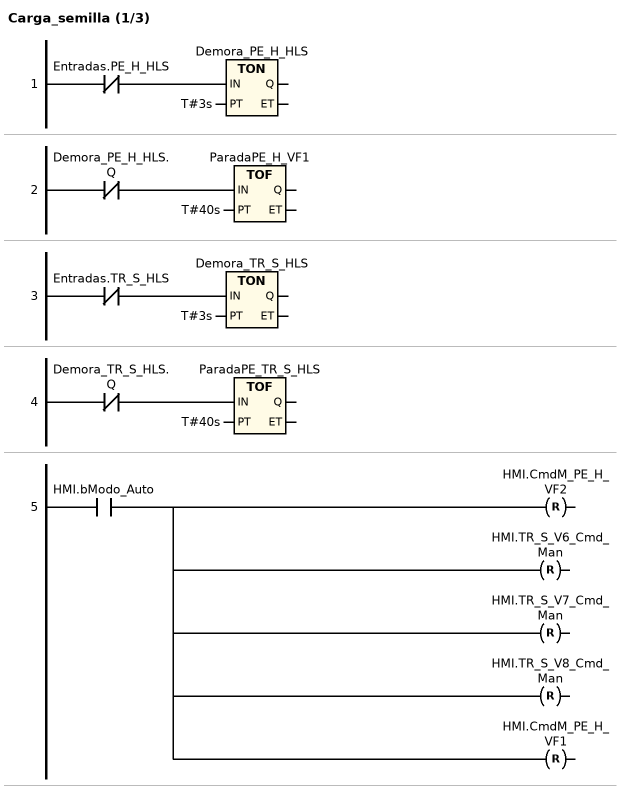
// NETWORK 1
Demora_PE_H_HLS(IN := NOT Entradas.PE_H_HLS, PT := T#3s); // TON

// NETWORK 2
ParadaPE_H_VF1(IN := NOT Demora_PE_H_HLS.Q, PT := T#40s); // TOF

// NETWORK 3
Demora_TR_S_HLS(IN := NOT Entradas.TR_S_HLS, PT := T#3s); // TON

// NETWORK 4
ParadaPE_TR_S_HLS(IN := NOT Demora_TR_S_HLS.Q, PT := T#40s); // TOF

// NETWORK 5
_w1 := HMI.bModo_Auto;
HMI.CmdM_PE_H_VF2 R= _w1;
HMI.TR_S_V6_Cmd_Man R= _w1;
HMI.TR_S_V7_Cmd_Man R= _w1;
HMI.TR_S_V8_Cmd_Man R= _w1;
HMI.CmdM_PE_H_VF1 R= _w1;

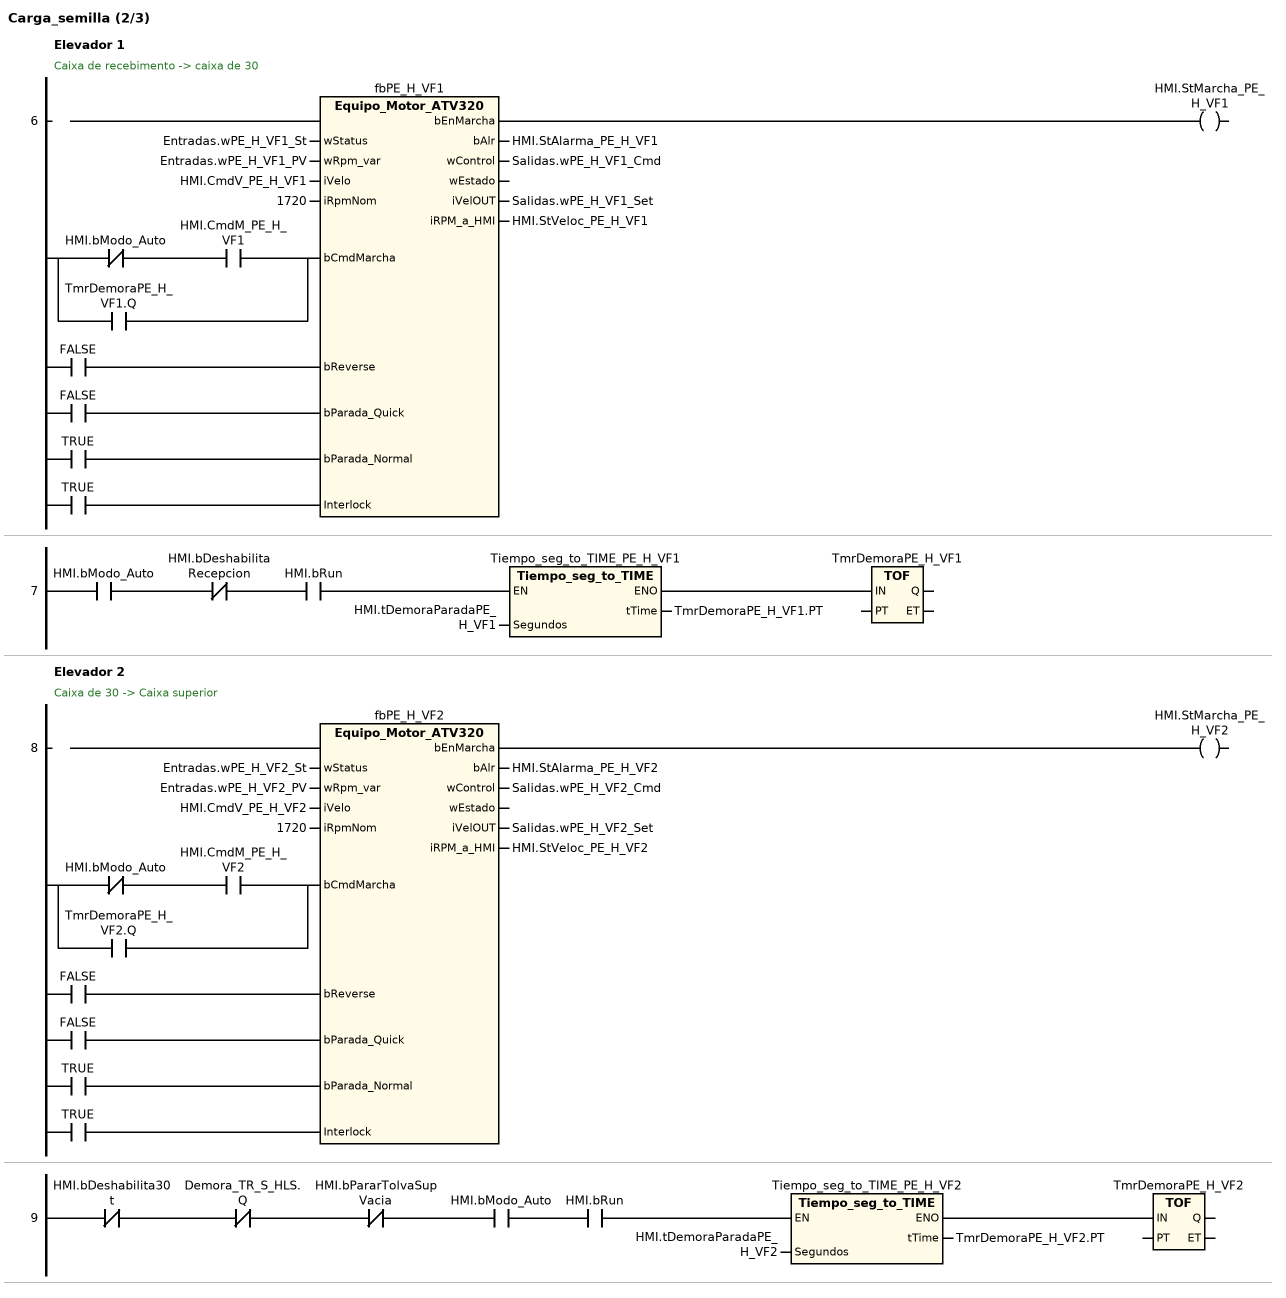
// NETWORK 6: Elevador 1
// Caixa de recebimento -> caixa de 30
fbPE_H_VF1(
    wStatus := Entradas.wPE_H_VF1_St,
    wRpm_var := Entradas.wPE_H_VF1_PV,
    iVelo := HMI.CmdV_PE_H_VF1,
    iRpmNom := 1720,
    bCmdMarcha := NOT HMI.bModo_Auto AND HMI.CmdM_PE_H_VF1 OR TmrDemoraPE_H_VF1.Q,
    bReverse := FALSE,
    bParada_Quick := FALSE,
    bParada_Normal := TRUE,
    Interlock := TRUE,
    bAlr => HMI.StAlarma_PE_H_VF1,
    wControl => Salidas.wPE_H_VF1_Cmd,
    iVelOUT => Salidas.wPE_H_VF1_Set,
    iRPM_a_HMI => HMI.StVeloc_PE_H_VF1); // Equipo_Motor_ATV320
HMI.StMarcha_PE_H_VF1 := fbPE_H_VF1.bEnMarcha;

// NETWORK 7
_w2 := HMI.bModo_Auto AND NOT HMI.bDeshabilitaRecepcion AND HMI.bRun;
IF _w2 THEN
    Tiempo_seg_to_TIME_PE_H_VF1(Segundos := HMI.tDemoraParadaPE_H_VF1, tTime => TmrDemoraPE_H_VF1.PT); // Tiempo_seg_to_TIME
END_IF
TmrDemoraPE_H_VF1(IN := _w2); // TOF

// NETWORK 8: Elevador 2
// Caixa de 30 -> Caixa superior
fbPE_H_VF2(
    wStatus := Entradas.wPE_H_VF2_St,
    wRpm_var := Entradas.wPE_H_VF2_PV,
    iVelo := HMI.CmdV_PE_H_VF2,
    iRpmNom := 1720,
    bCmdMarcha := NOT HMI.bModo_Auto AND HMI.CmdM_PE_H_VF2 OR TmrDemoraPE_H_VF2.Q,
    bReverse := FALSE,
    bParada_Quick := FALSE,
    bParada_Normal := TRUE,
    Interlock := TRUE,
    bAlr => HMI.StAlarma_PE_H_VF2,
    wControl => Salidas.wPE_H_VF2_Cmd,
    iVelOUT => Salidas.wPE_H_VF2_Set,
    iRPM_a_HMI => HMI.StVeloc_PE_H_VF2); // Equipo_Motor_ATV320
HMI.StMarcha_PE_H_VF2 := fbPE_H_VF2.bEnMarcha;

// NETWORK 9
_w3 := NOT HMI.bDeshabilita30t AND NOT Demora_TR_S_HLS.Q AND NOT HMI.bPararTolvaSupVacia AND HMI.bModo_Auto AND HMI.bRun;
IF _w3 THEN
    Tiempo_seg_to_TIME_PE_H_VF2(Segundos := HMI.tDemoraParadaPE_H_VF2, tTime => TmrDemoraPE_H_VF2.PT); // Tiempo_seg_to_TIME
END_IF
TmrDemoraPE_H_VF2(IN := _w3); // TOF

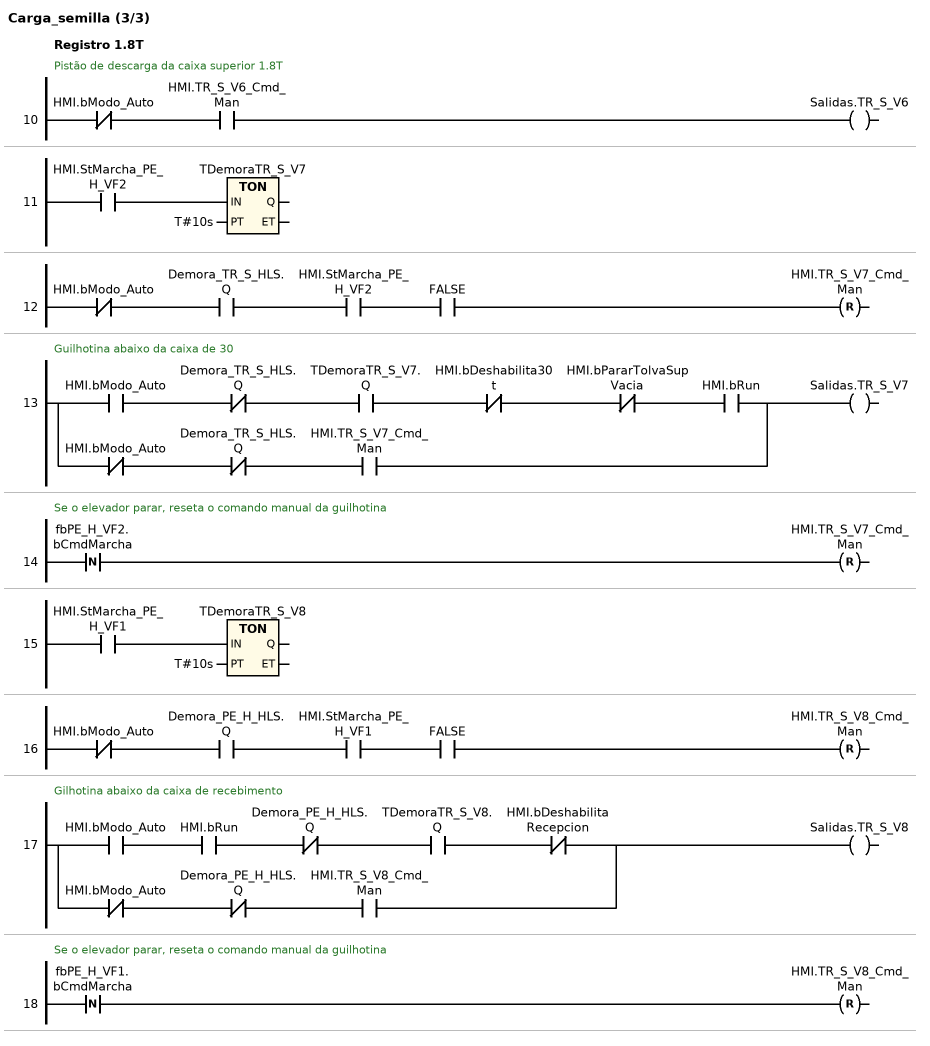
// NETWORK 10: Registro 1.8T
// Pistão de descarga da caixa superior 1.8T
Salidas.TR_S_V6 := NOT HMI.bModo_Auto AND HMI.TR_S_V6_Cmd_Man;

// NETWORK 11
TDemoraTR_S_V7(IN := HMI.StMarcha_PE_H_VF2, PT := T#10s); // TON

// NETWORK 12
HMI.TR_S_V7_Cmd_Man R= NOT HMI.bModo_Auto AND Demora_TR_S_HLS.Q AND HMI.StMarcha_PE_H_VF2 AND FALSE;

// NETWORK 13
// Guilhotina abaixo da caixa de 30
Salidas.TR_S_V7 := HMI.bModo_Auto AND NOT Demora_TR_S_HLS.Q AND TDemoraTR_S_V7.Q AND NOT HMI.bDeshabilita30t AND NOT HMI.bPararTolvaSupVacia AND HMI.bRun OR NOT HMI.bModo_Auto AND NOT Demora_TR_S_HLS.Q AND HMI.TR_S_V7_Cmd_Man;

// NETWORK 14
// Se o elevador parar, reseta o comando manual da guilhotina
_ft1(CLK := fbPE_H_VF2.bCmdMarcha);
HMI.TR_S_V7_Cmd_Man R= _ft1.Q;

// NETWORK 15
TDemoraTR_S_V8(IN := HMI.StMarcha_PE_H_VF1, PT := T#10s); // TON

// NETWORK 16
HMI.TR_S_V8_Cmd_Man R= NOT HMI.bModo_Auto AND Demora_PE_H_HLS.Q AND HMI.StMarcha_PE_H_VF1 AND FALSE;

// NETWORK 17
// Gilhotina abaixo da caixa de recebimento
Salidas.TR_S_V8 := HMI.bModo_Auto AND HMI.bRun AND NOT Demora_PE_H_HLS.Q AND TDemoraTR_S_V8.Q AND NOT HMI.bDeshabilitaRecepcion OR NOT HMI.bModo_Auto AND NOT Demora_PE_H_HLS.Q AND HMI.TR_S_V8_Cmd_Man;

// NETWORK 18
// Se o elevador parar, reseta o comando manual da guilhotina
_ft2(CLK := fbPE_H_VF1.bCmdMarcha);
HMI.TR_S_V8_Cmd_Man R= _ft2.Q;

END_PROGRAM

// ---- POUs/Polvo 1/Dosificador_Polvo_1.TcPOU
PROGRAM Dosificador_Polvo_1
VAR
	fbDosificador_P1 :Equipo_Motor_ATV320;
	Balanza_P1_WT1: Balanza;
	fbTR_P1_VI: Equipo_Motor_ATV320;
	TararP1:BOOL;
	dHS:DINT;
	
	Tmr_Alr_ZeroSpeed: TON;
	TDemoraInyectarPolvo: TON;
	Tiempo_seg_to_TIME_TDemoraInyec: Tiempo_seg_to_TIME;
	Auxtdemora: TIME;
	Calc_Veloc_Polvo_1: Calc_Veloc_Polvo;
	Calc_Veloc_Polvo_1i: Calc_Veloc_Polvo;
	Tiempo_seg_to_TIME_TInyeccion: Tiempo_seg_to_TIME;
	AuxInyec: TIME;
	TInyeccion: TON;
	ModoCalibrarP1 :BOOL;
	
	InyectarCalibrarP1: BOOL;
	Calibracion_Po_calc_P1: Calibracion_Po_calc;
	PolvoAsociado:STRING;
	TR_P1_WT1_rValue_REAL: REAL;
	TON_SolicitaPo: TON;
END_VAR
VAR PERSISTENT
	UltimaCalibracao	:UDINT;	//Data da ultima calibração feita com sucesso
END_VAR
VAR // added by the converter: edge detectors and wires of the graphical bodies
    _w1, _w2, _w3 : BOOL;
    _ft1 : F_TRIG;
    _rt1 : R_TRIG;
END_VAR

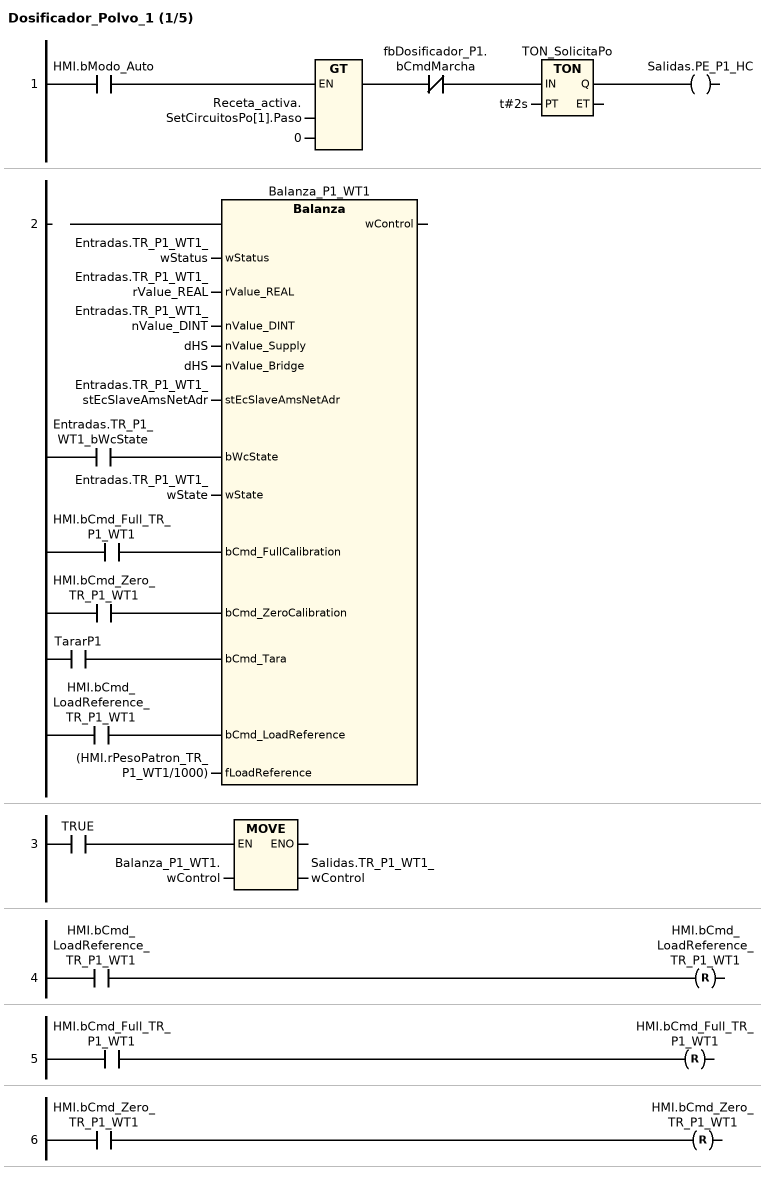
// NETWORK 1
TON_SolicitaPo(IN := (HMI.bModo_Auto AND Receta_activa.SetCircuitosPo[1].Paso > 0) AND NOT fbDosificador_P1.bCmdMarcha, PT := t#2s); // TON
Salidas.PE_P1_HC := TON_SolicitaPo.Q;

// NETWORK 2
Balanza_P1_WT1(
    wStatus := Entradas.TR_P1_WT1_wStatus,
    rValue_REAL := Entradas.TR_P1_WT1_rValue_REAL,
    nValue_DINT := Entradas.TR_P1_WT1_nValue_DINT,
    nValue_Supply := dHS,
    nValue_Bridge := dHS,
    stEcSlaveAmsNetAdr := Entradas.TR_P1_WT1_stEcSlaveAmsNetAdr,
    bWcState := Entradas.TR_P1_WT1_bWcState,
    wState := Entradas.TR_P1_WT1_wState,
    bCmd_FullCalibration := HMI.bCmd_Full_TR_P1_WT1,
    bCmd_ZeroCalibration := HMI.bCmd_Zero_TR_P1_WT1,
    bCmd_Tara := TararP1,
    bCmd_LoadReference := HMI.bCmd_LoadReference_TR_P1_WT1,
    fLoadReference := (HMI.rPesoPatron_TR_P1_WT1/1000)); // Balanza

// NETWORK 3
Salidas.TR_P1_WT1_wControl := Balanza_P1_WT1.wControl;

// NETWORK 4
HMI.bCmd_LoadReference_TR_P1_WT1 R= HMI.bCmd_LoadReference_TR_P1_WT1;

// NETWORK 5
HMI.bCmd_Full_TR_P1_WT1 R= HMI.bCmd_Full_TR_P1_WT1;

// NETWORK 6
HMI.bCmd_Zero_TR_P1_WT1 R= HMI.bCmd_Zero_TR_P1_WT1;

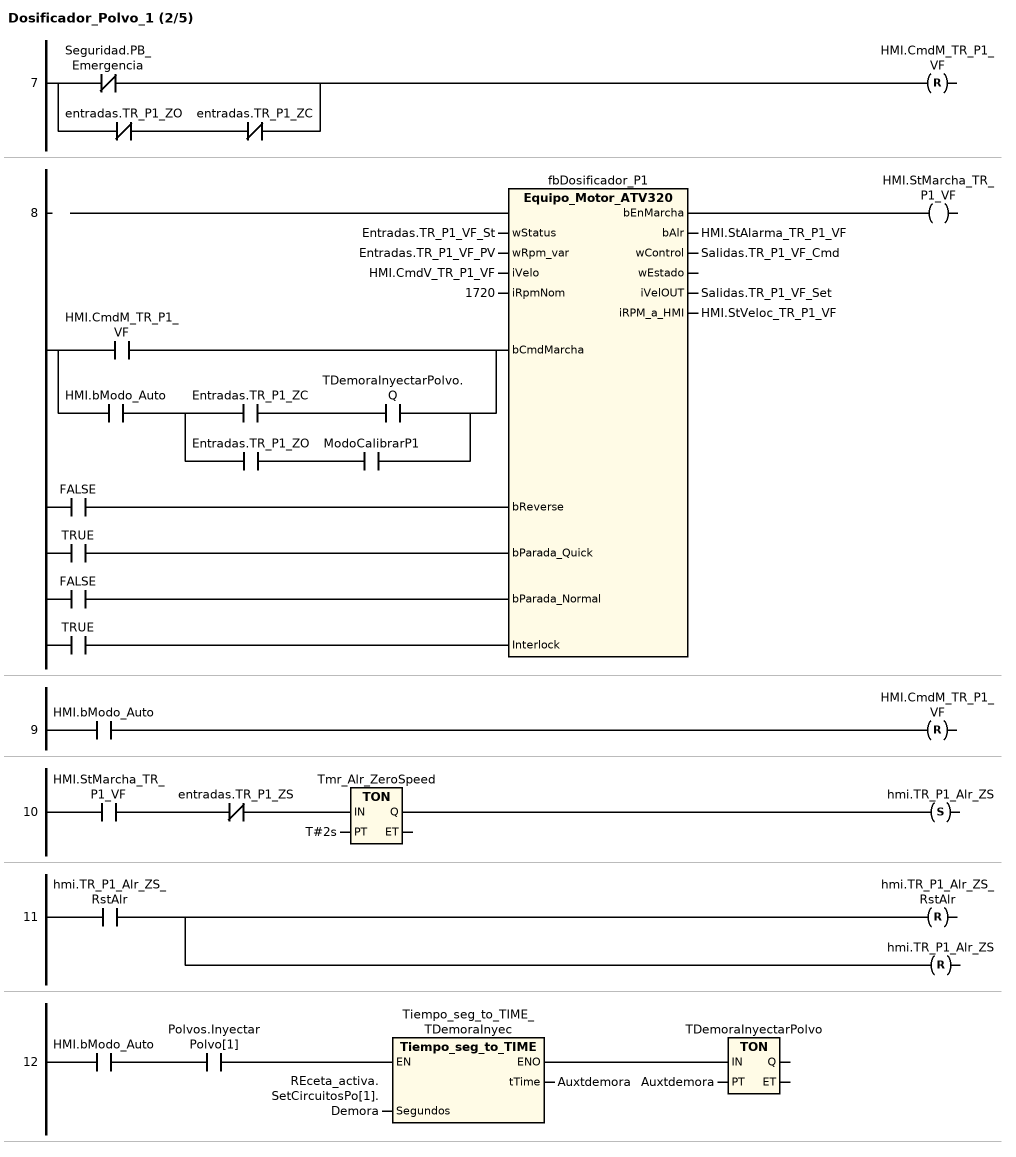
// NETWORK 7
HMI.CmdM_TR_P1_VF R= NOT Seguridad.PB_Emergencia OR NOT entradas.TR_P1_ZO AND NOT entradas.TR_P1_ZC;

// NETWORK 8
fbDosificador_P1(
    wStatus := Entradas.TR_P1_VF_St,
    wRpm_var := Entradas.TR_P1_VF_PV,
    iVelo := HMI.CmdV_TR_P1_VF,
    iRpmNom := 1720,
    bCmdMarcha := HMI.CmdM_TR_P1_VF OR HMI.bModo_Auto AND (Entradas.TR_P1_ZC AND TDemoraInyectarPolvo.Q OR Entradas.TR_P1_ZO AND ModoCalibrarP1),
    bReverse := FALSE,
    bParada_Quick := TRUE,
    bParada_Normal := FALSE,
    Interlock := TRUE,
    bAlr => HMI.StAlarma_TR_P1_VF,
    wControl => Salidas.TR_P1_VF_Cmd,
    iVelOUT => Salidas.TR_P1_VF_Set,
    iRPM_a_HMI => HMI.StVeloc_TR_P1_VF); // Equipo_Motor_ATV320
HMI.StMarcha_TR_P1_VF := fbDosificador_P1.bEnMarcha;

// NETWORK 9
HMI.CmdM_TR_P1_VF R= HMI.bModo_Auto;

// NETWORK 10
Tmr_Alr_ZeroSpeed(IN := HMI.StMarcha_TR_P1_VF AND NOT entradas.TR_P1_ZS, PT := T#2s); // TON
hmi.TR_P1_Alr_ZS S= Tmr_Alr_ZeroSpeed.Q;

// NETWORK 11
_w1 := hmi.TR_P1_Alr_ZS_RstAlr;
hmi.TR_P1_Alr_ZS_RstAlr R= _w1;
hmi.TR_P1_Alr_ZS R= _w1;

// NETWORK 12
_w2 := HMI.bModo_Auto AND Polvos.InyectarPolvo[1];
IF _w2 THEN
    Tiempo_seg_to_TIME_TDemoraInyec(Segundos := REceta_activa.SetCircuitosPo[1].Demora, tTime => Auxtdemora); // Tiempo_seg_to_TIME
END_IF
TDemoraInyectarPolvo(IN := _w2, PT := Auxtdemora); // TON

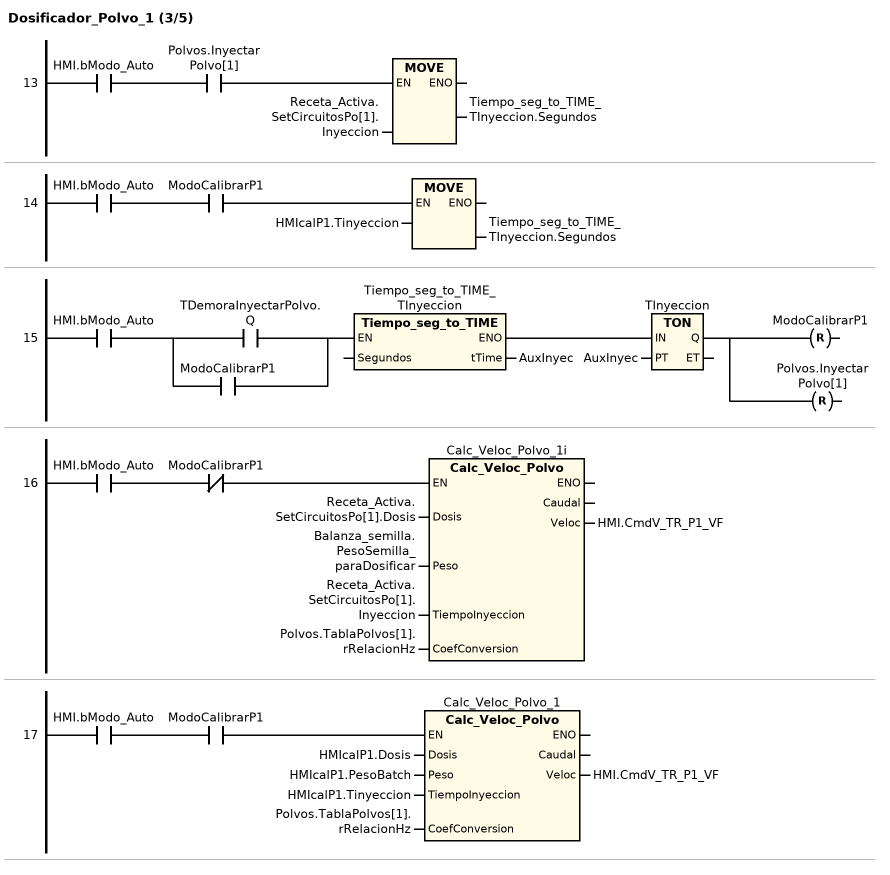
// NETWORK 13
IF HMI.bModo_Auto AND Polvos.InyectarPolvo[1] THEN
    Tiempo_seg_to_TIME_TInyeccion.Segundos := Receta_Activa.SetCircuitosPo[1].Inyeccion;
END_IF

// NETWORK 14
IF HMI.bModo_Auto AND ModoCalibrarP1 THEN Tiempo_seg_to_TIME_TInyeccion.Segundos := HMIcalP1.Tinyeccion; END_IF

// NETWORK 15
_w3 := HMI.bModo_Auto AND (TDemoraInyectarPolvo.Q OR ModoCalibrarP1);
IF _w3 THEN
    Tiempo_seg_to_TIME_TInyeccion(tTime => AuxInyec); // Tiempo_seg_to_TIME
END_IF
TInyeccion(IN := _w3, PT := AuxInyec); // TON
ModoCalibrarP1 R= TInyeccion.Q;
Polvos.InyectarPolvo[1] R= TInyeccion.Q;

// NETWORK 16
IF HMI.bModo_Auto AND NOT ModoCalibrarP1 THEN
    Calc_Veloc_Polvo_1i(
        Dosis := Receta_Activa.SetCircuitosPo[1].Dosis,
        Peso := Balanza_semilla.PesoSemilla_paraDosificar,
        TiempoInyeccion := Receta_Activa.SetCircuitosPo[1].Inyeccion,
        CoefConversion := Polvos.TablaPolvos[1].rRelacionHz,
        Veloc => HMI.CmdV_TR_P1_VF); // Calc_Veloc_Polvo
END_IF

// NETWORK 17
IF HMI.bModo_Auto AND ModoCalibrarP1 THEN
    Calc_Veloc_Polvo_1(
        Dosis := HMIcalP1.Dosis,
        Peso := HMIcalP1.PesoBatch,
        TiempoInyeccion := HMIcalP1.Tinyeccion,
        CoefConversion := Polvos.TablaPolvos[1].rRelacionHz,
        Veloc => HMI.CmdV_TR_P1_VF); // Calc_Veloc_Polvo
END_IF

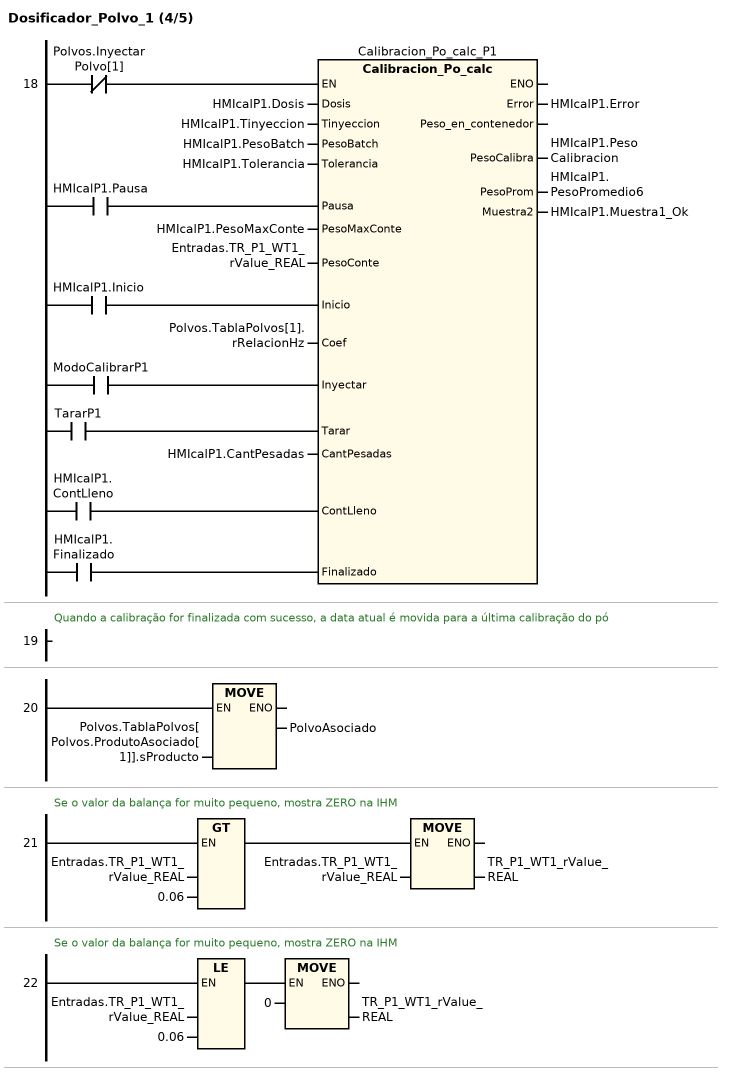
// NETWORK 18
IF NOT Polvos.InyectarPolvo[1] THEN
    Calibracion_Po_calc_P1(
        Dosis := HMIcalP1.Dosis,
        Tinyeccion := HMIcalP1.Tinyeccion,
        PesoBatch := HMIcalP1.PesoBatch,
        Tolerancia := HMIcalP1.Tolerancia,
        Pausa := HMIcalP1.Pausa,
        PesoMaxConte := HMIcalP1.PesoMaxConte,
        PesoConte := Entradas.TR_P1_WT1_rValue_REAL,
        Inicio := HMIcalP1.Inicio,
        Coef := Polvos.TablaPolvos[1].rRelacionHz,
        Inyectar := ModoCalibrarP1,
        Tarar := TararP1,
        CantPesadas := HMIcalP1.CantPesadas,
        ContLleno := HMIcalP1.ContLleno,
        Finalizado := HMIcalP1.Finalizado,
        Error => HMIcalP1.Error,
        PesoCalibra => HMIcalP1.PesoCalibracion,
        PesoProm => HMIcalP1.PesoPromedio6,
        Muestra2 => HMIcalP1.Muestra1_Ok); // Calibracion_Po_calc
END_IF

// NETWORK 19
// Quando a calibração for finalizada com sucesso, a data atual é movida para a última calibração do pó

// NETWORK 20
PolvoAsociado := Polvos.TablaPolvos[Polvos.ProdutoAsociado[1]].sProducto;

// NETWORK 21
// Se o valor da balança for muito pequeno, mostra ZERO na IHM
IF Entradas.TR_P1_WT1_rValue_REAL > 0.06 THEN TR_P1_WT1_rValue_REAL := Entradas.TR_P1_WT1_rValue_REAL; END_IF

// NETWORK 22
// Se o valor da balança for muito pequeno, mostra ZERO na IHM
IF Entradas.TR_P1_WT1_rValue_REAL <= 0.06 THEN TR_P1_WT1_rValue_REAL := 0; END_IF

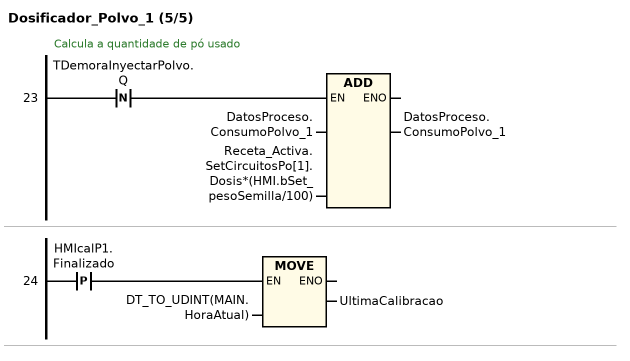
// NETWORK 23
// Calcula a quantidade de pó usado
_ft1(CLK := TDemoraInyectarPolvo.Q);
IF _ft1.Q THEN
    DatosProceso.ConsumoPolvo_1 := DatosProceso.ConsumoPolvo_1 + (Receta_Activa.SetCircuitosPo[1].Dosis*(HMI.bSet_pesoSemilla/100));
END_IF

// NETWORK 24
_rt1(CLK := HMIcalP1.Finalizado);
IF _rt1.Q THEN UltimaCalibracao := DT_TO_UDINT(MAIN.HoraAtual); END_IF

END_PROGRAM

// ---- POUs/Elementos/Calc_Veloc_Polvo.TcPOU
FUNCTION_BLOCK Calc_Veloc_Polvo
VAR_INPUT
	Dosis:REAL;//gr/100 Kg
	Peso:REAL;// 100 Kg
	TiempoInyeccion:DINT;// seg
	CoefConversion:REAL;
END_VAR
VAR_OUTPUT
	Caudal:REAL;//grs/seg
	Veloc:REAL;//
END_VAR
VAR
END_VAR

IF TiempoInyeccion=0 THEN
	TiempoInyeccion:=1;
END_IF
Caudal:= Dosis * Peso/100 / DINT_TO_REAL (TiempoInyeccion);
Veloc:=Caudal*CoefConversion;

END_FUNCTION_BLOCK

// ---- POUs/Elementos/Calibracion_Po_calc.TcPOU
FUNCTION_BLOCK Calibracion_Po_calc
VAR_INPUT
	Dosis:REAL;
	Tinyeccion:DINT;
	PesoBatch:REAL;
	Tolerancia:REAL;
	Pausa:BOOL;
	PesoMaxConte:REAL;
	PesoConte:REAL;
END_VAR
VAR_OUTPUT
	Error:REAL;
	Peso_en_contenedor:REAL;
	PesoCalibra:REAL;
	PesoProm:REAL;
    Muestra2:BOOL;
END_VAR
VAR_IN_OUT
	Inicio:BOOL;
	Coef:REAL;
	Inyectar:BOOL;
	Tarar:BOOL;
	CantPesadas:INT;
	ContLleno:BOOL;
	Finalizado:BOOL;	
END_VAR
VAR

	IniciarCal: R_TRIG;
	Caudal:REAL;
	PesoMax:REAL;
	PesoMin:REAL;
	Calibrando:BOOL;
	IniInyectar:R_TRIG;
	FinInyectar:F_TRIG;
	Inyectando:BOOL;
	PesoIni:REAL;
	Pesada:ARRAY [1..6]OF REAL;
	Muestra1:BOOL;
	PromMuestra:REAL;
	IniCal:BOOL;
	IniIny:BOOL;
	FinIny:BOOL;
	tDemoraFinIny:TON;
	tDemoraFinIny2:TON;
	StepCal:INT;
	bContenedorLleno:F_TRIG;
	borrarContenedorLleno:BOOL;
	CancelarCal:F_TRIG;
	CanCal: BOOL;
	Teste: INT;
	i: INT;
	PromMuestra2: REAL;
END_VAR


IniciarCal(CLK:=Inicio , Q=>IniCal );
IF IniCal THEN
	StepCal:=1;
	IniCal:=0;
END_IF
CancelarCal(CLK:=Inicio , Q=>CanCal );

IF CanCal  THEN
	StepCal:=0;
	Pausa:=FALSE;
	CantPesadas:=0;
	Calibrando:=FALSE;
	Muestra1:=FALSE;
	Muestra2:=FALSE;
	CanCal:=0;
END_IF
PesoCalibra:=Dosis*PesoBatch/100;
bContenedorLleno(CLK:=ContLleno ,Q=>borrarContenedorLleno );
IF borrarContenedorLleno THEN
	Peso_en_contenedor:=0;
	Tarar:=TRUE;
	borrarContenedorLleno:=0;
END_IF

CASE StepCal OF
	1: 
		IF Tinyeccion=0 THEN
			Tinyeccion:=1;
		END_IF
		Tarar:=TRUE;
		Caudal:=PesoCalibra/DINT_TO_REAL (Tinyeccion);
		PesoMax:=(PesoCalibra*(1+Tolerancia/100))/1000;
		PesoMin:=(PesoCalibra*(1-Tolerancia/100))/1000;
		Pesada[1]:=0;
		Pesada[2]:=0;
		Pesada[3]:=0;
		Pesada[4]:=0;
		Pesada[5]:=0;
		Pesada[6]:=0;
		Finalizado:=0;
		Peso_en_contenedor:=0;
		CantPesadas:=0;
		Calibrando:=TRUE;
		IniCal:=0;
		StepCal:=2;
		
	2: 	Inyectar:=TRUE;
		Muestra1:=TRUE;
		//Tarar:=FALSE;
		PesoIni:=PesoConte;
		StepCal:=3;
		
	3: 	tDemoraFinIny(IN:=NOT Inyectar,PT:=T#10S);;
		IF tDemoraFinIny.Q THEN
			Tarar:=FALSE;
			StepCal:=4;
		END_IF
		
	4: 	CantPesadas := CantPesadas + 1;	
		Pesada[CantPesadas] := PesoConte - PesoIni;
		Peso_en_contenedor := Peso_en_contenedor + Pesada[CantPesadas];
		StepCal := 5;
		
	5:	IF Peso_en_contenedor > (0.9 * PesoMaxConte) THEN
			ContLleno:=1;
		ELSE
			StepCal:=6;		
		END_IF;
		
	6:		IF CantPesadas<3 THEN
				IF NOT Pausa THEN
					StepCal:=2;
				END_IF
			ELSE
				StepCal:=7;	
			END_IF;
	
	7://Calculo error muestra1
		IF CantPesadas=3 AND Muestra1 AND NOT Muestra2 AND NOT Inyectar THEN
			PromMuestra:=(Pesada[1]+Pesada[2]+Pesada[3])/3;
			IF (PromMuestra<=PesoMax) AND (PromMuestra>=PesoMin) THEN
				Muestra2:=TRUE;
				StepCal:=8;	
			ELSE
				//Coef:=Coef*	(PesoCalibra*0.001)/PromMuestra;
				
				IF PesoCalibra / (PromMuestra * 1000) >= 3 THEN
					Teste := 1;
					Coef := Coef + 0.4;
				ELSIF PesoCalibra / (PromMuestra * 1000) < 3 AND PesoCalibra / (PromMuestra * 1000) >= 2 THEN
					Teste := 2;
					Coef := Coef + 0.03;
				ELSIF PesoCalibra / (PromMuestra * 1000) < 2 AND PesoCalibra / (PromMuestra * 1000) >= 1 THEN
					Teste := 3;
					Coef := Coef + 0.03;
				ELSIF PesoCalibra / (PromMuestra * 1000) < 1 AND PesoCalibra / (PromMuestra * 1000) >= 0.5 THEN
					Teste := 4;
					Coef := Coef - 0.03;
				ELSE
					Coef := Coef - 0.1;
					Teste := 5;
				END_IF
				//Coef:=Coef+((((PesoCalibra*0.001)-PromMuestra)/(PesoCalibra*0.001))/1);
				Muestra1:=FALSE;
				CantPesadas:=0;	
				StepCal:=2;	
			FOR i := 1 TO 6 DO
				Pesada[i] := 0;
			END_FOR		
			END_IF		
		END_IF;
		
	8:	Inyectar:=TRUE;
		PesoIni:=PesoConte;
		StepCal:=9;
		
	9:	tDemoraFinIny2(IN:=NOT Inyectar,PT:=T#10S);;
		IF tDemoraFinIny2.Q THEN
			StepCal:=10;
		END_IF;
		
	10:	CantPesadas:=CantPesadas+1;	
		Pesada[CantPesadas]:=PesoConte-PesoIni;
		Peso_en_contenedor:=Peso_en_contenedor+Pesada[CantPesadas];
		StepCal:=11;
		
	11:	IF Peso_en_contenedor>(0.9*PesoMaxConte) THEN
			ContLleno:=1;
		ELSE
			StepCal:=12;		
		END_IF;
			
	12:		IF CantPesadas<6 THEN
				IF NOT Pausa THEN
					StepCal:=8;
				END_IF	
			ELSE
				StepCal:=13;	
			END_IF;
	
	13:	
			PromMuestra2:=(Pesada[4]+Pesada[5]+Pesada[6])/3;
		IF ((PromMuestra2<PesoMax) AND (PromMuestra2>PesoMin)) THEN
			PesoProm:=((Pesada[1]+Pesada[2]+Pesada[3]+Pesada[4]+Pesada[5]+Pesada[6])/6)*1000;
			Error:=((PesoCalibra-PesoProm)/PesoCalibra)*100;
			Inicio:=FALSE;
			Muestra1:=FALSE;
			Muestra2:=FALSE;
			Calibrando:=FALSE;
			Finalizado:=TRUE;
			Tarar:=0;
			StepCal:=0;	
		ELSE
			//Coef:=Coef+((((PesoCalibra*0.001)-PromMuestra)/(PesoCalibra*0.001))/100);
			//Coef:=Coef*(PesoCalibra*0.001)/PromMuestra;
			IF PesoCalibra / (PromMuestra * 1000) >= 3 THEN
				Coef := Coef + 0.4;
			ELSIF PesoCalibra / (PromMuestra * 1000) < 3 AND PesoCalibra / (PromMuestra * 1000) >= 2 THEN
				Coef := Coef + 0.03;
			ELSIF PesoCalibra / (PromMuestra * 1000) < 2 AND PesoCalibra / (PromMuestra * 1000) >= 1 THEN
				Coef := Coef + 0.03;
			ELSIF PesoCalibra / (PromMuestra * 1000) < 1 AND PesoCalibra / (PromMuestra * 1000) >= 0.5 THEN
				Coef := Coef - 0.03;
			ELSE
				Coef := Coef - 0.1;
			END_IF
			Muestra1:=FALSE;
			Muestra2:=FALSE;
			CantPesadas:=0;
			StepCal:=2;	
			FOR i := 1 TO 6 DO
				Pesada[i] := 0;
			END_FOR
		END_IF;		
		
END_CASE

//Faz a média de valores de acordo com a contagem de pesagens
IF CantPesadas > 0 THEN
	//PromMuestra:=(Pesada[1]+Pesada[2]+Pesada[3]+Pesada[4]+Pesada[5]+Pesada[6])/CantPesadas;
	PromMuestra := 0;
	FOR i := 1 TO CantPesadas DO
		PromMuestra := PromMuestra + (Pesada[i]/CantPesadas);
	END_FOR
END_IF;

//Verifica se o recipiente está cheio
IF Peso_en_contenedor>(0.9*PesoMaxConte) THEN
	ContLleno:=1;
END_IF;

END_FUNCTION_BLOCK

// ---- POUs/Inicio.TcPOU
PROGRAM Inicio
VAR
	Premarcha: BOOL;
	TmrPremarcha: TON;
END_VAR
VAR // added by the converter: edge detectors and wires of the graphical bodies
    _rt1 : R_TRIG;
    _w1, _w2 : BOOL;
END_VAR

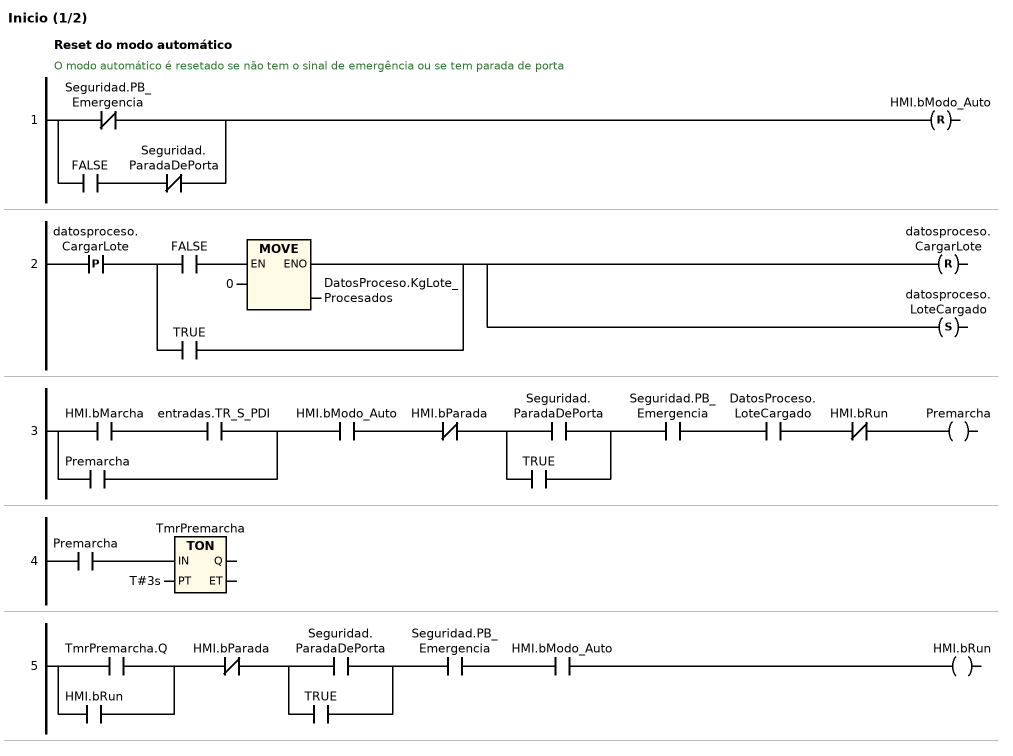
// NETWORK 1: Reset do modo automático
// O modo automático é resetado se não tem o sinal de emergência ou se tem parada de porta
HMI.bModo_Auto R= NOT Seguridad.PB_Emergencia OR FALSE AND NOT Seguridad.ParadaDePorta;

// NETWORK 2
_rt1(CLK := datosproceso.CargarLote);
_w1 := _rt1.Q AND TRUE;
IF NOT _w1 THEN
    _w2 := _rt1.Q AND FALSE;
    IF _w2 THEN DatosProceso.KgLote_Procesados := 0; END_IF
    _w1 := _w2;
END_IF
datosproceso.CargarLote R= _w1;
datosproceso.LoteCargado S= _w1;

// NETWORK 3
Premarcha := (HMI.bMarcha AND entradas.TR_S_PDI OR Premarcha) AND HMI.bModo_Auto AND NOT HMI.bParada AND (Seguridad.ParadaDePorta OR TRUE) AND Seguridad.PB_Emergencia AND DatosProceso.LoteCargado AND NOT HMI.bRun;

// NETWORK 4
TmrPremarcha(IN := Premarcha, PT := T#3s); // TON

// NETWORK 5
HMI.bRun := (TmrPremarcha.Q OR HMI.bRun) AND NOT HMI.bParada AND (Seguridad.ParadaDePorta OR TRUE) AND Seguridad.PB_Emergencia AND HMI.bModo_Auto;

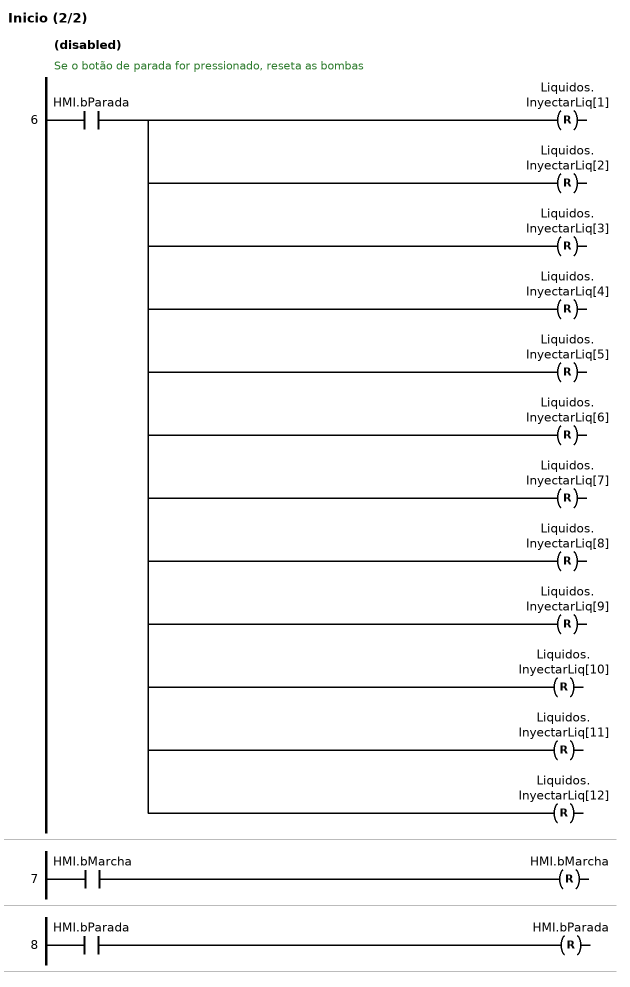
// NETWORK 6 (disabled)
// Se o botão de parada for pressionado, reseta as bombas
// Liquidos.InyectarLiq[1] R= HMI.bParada;
// Liquidos.InyectarLiq[2] R= HMI.bParada;
// Liquidos.InyectarLiq[3] R= HMI.bParada;
// Liquidos.InyectarLiq[4] R= HMI.bParada;
// Liquidos.InyectarLiq[5] R= HMI.bParada;
// Liquidos.InyectarLiq[6] R= HMI.bParada;
// Liquidos.InyectarLiq[7] R= HMI.bParada;
// Liquidos.InyectarLiq[8] R= HMI.bParada;
// Liquidos.InyectarLiq[9] R= HMI.bParada;
// Liquidos.InyectarLiq[10] R= HMI.bParada;
// Liquidos.InyectarLiq[11] R= HMI.bParada;
// Liquidos.InyectarLiq[12] R= HMI.bParada;

// NETWORK 7
HMI.bMarcha R= HMI.bMarcha;

// NETWORK 8
HMI.bParada R= HMI.bParada;

END_PROGRAM

// ---- POUs/Polvo 2/Dosificador_Polvo_2.TcPOU
PROGRAM Dosificador_Polvo_2
VAR
	fbDosificador_P2 :Equipo_Motor_ATV320;
	Balanza_P2_WT1: Balanza;
	fbTR_P2_VI: Equipo_Motor_ATV320;
	TararP2:BOOL;
	dHS:DINT;
	
	Tmr_Alr_ZeroSpeed: TON;
	TDemoraInyectarPolvo: TON;
	Tiempo_seg_to_TIME_TDemoraInyec: Tiempo_seg_to_TIME;
	Auxtdemora: TIME;
	Calc_Veloc_Polvo_2: Calc_Veloc_Polvo;
	Tiempo_seg_to_TIME_TInyeccion: Tiempo_seg_to_TIME;
	AuxInyec: TIME;
	TInyeccion: TON;
	ModoCalibrarP2 :BOOL;
	
	InyectarCalibrarP2: BOOL;
	Calibracion_Po_calc_P2: Calibracion_Po_calc;
	PolvoAsociado:STRING;
	TR_P2_WT1_rValue_REAL: REAL;
	TON_SolicitaPo: TON;
END_VAR
VAR PERSISTENT
	UltimaCalibracao	:UDINT;	//Data da ultima calibração feita com sucesso
END_VAR
VAR // added by the converter: edge detectors and wires of the graphical bodies
    _w1, _w2, _w3 : BOOL;
    _ft1 : F_TRIG;
    _rt1 : R_TRIG;
END_VAR

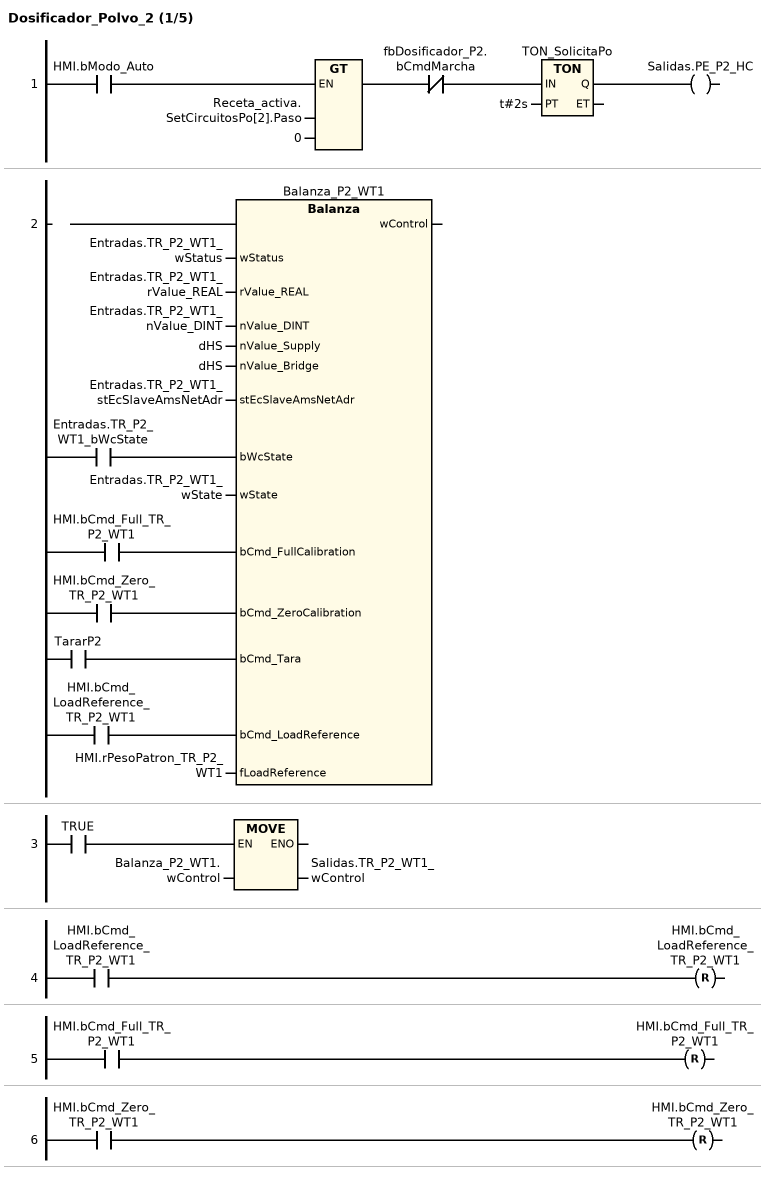
// NETWORK 1
TON_SolicitaPo(IN := (HMI.bModo_Auto AND Receta_activa.SetCircuitosPo[2].Paso > 0) AND NOT fbDosificador_P2.bCmdMarcha, PT := t#2s); // TON
Salidas.PE_P2_HC := TON_SolicitaPo.Q;

// NETWORK 2
Balanza_P2_WT1(
    wStatus := Entradas.TR_P2_WT1_wStatus,
    rValue_REAL := Entradas.TR_P2_WT1_rValue_REAL,
    nValue_DINT := Entradas.TR_P2_WT1_nValue_DINT,
    nValue_Supply := dHS,
    nValue_Bridge := dHS,
    stEcSlaveAmsNetAdr := Entradas.TR_P2_WT1_stEcSlaveAmsNetAdr,
    bWcState := Entradas.TR_P2_WT1_bWcState,
    wState := Entradas.TR_P2_WT1_wState,
    bCmd_FullCalibration := HMI.bCmd_Full_TR_P2_WT1,
    bCmd_ZeroCalibration := HMI.bCmd_Zero_TR_P2_WT1,
    bCmd_Tara := TararP2,
    bCmd_LoadReference := HMI.bCmd_LoadReference_TR_P2_WT1,
    fLoadReference := HMI.rPesoPatron_TR_P2_WT1); // Balanza

// NETWORK 3
Salidas.TR_P2_WT1_wControl := Balanza_P2_WT1.wControl;

// NETWORK 4
HMI.bCmd_LoadReference_TR_P2_WT1 R= HMI.bCmd_LoadReference_TR_P2_WT1;

// NETWORK 5
HMI.bCmd_Full_TR_P2_WT1 R= HMI.bCmd_Full_TR_P2_WT1;

// NETWORK 6
HMI.bCmd_Zero_TR_P2_WT1 R= HMI.bCmd_Zero_TR_P2_WT1;

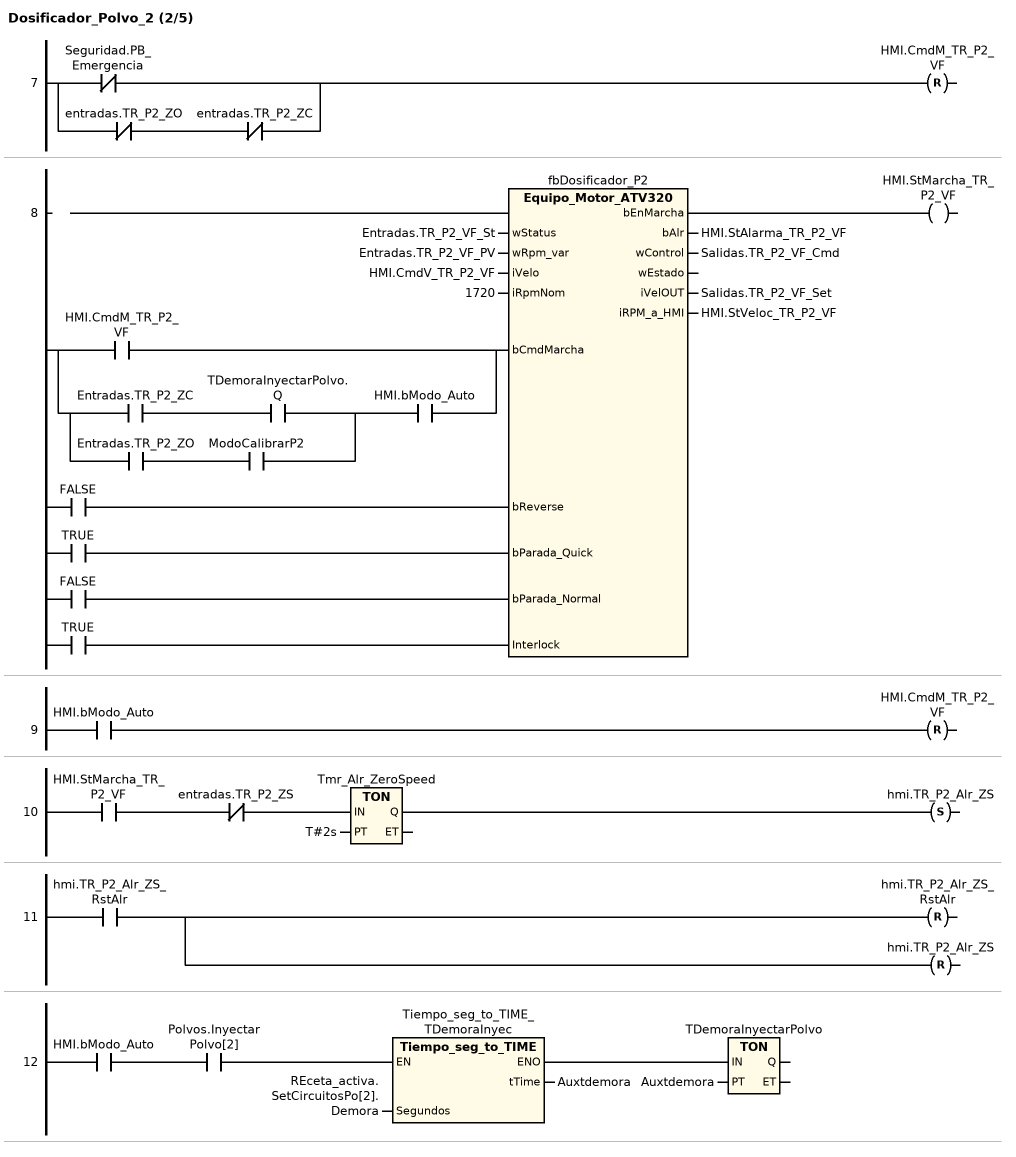
// NETWORK 7
HMI.CmdM_TR_P2_VF R= NOT Seguridad.PB_Emergencia OR NOT entradas.TR_P2_ZO AND NOT entradas.TR_P2_ZC;

// NETWORK 8
fbDosificador_P2(
    wStatus := Entradas.TR_P2_VF_St,
    wRpm_var := Entradas.TR_P2_VF_PV,
    iVelo := HMI.CmdV_TR_P2_VF,
    iRpmNom := 1720,
    bCmdMarcha := HMI.CmdM_TR_P2_VF OR (Entradas.TR_P2_ZC AND TDemoraInyectarPolvo.Q OR Entradas.TR_P2_ZO AND ModoCalibrarP2) AND HMI.bModo_Auto,
    bReverse := FALSE,
    bParada_Quick := TRUE,
    bParada_Normal := FALSE,
    Interlock := TRUE,
    bAlr => HMI.StAlarma_TR_P2_VF,
    wControl => Salidas.TR_P2_VF_Cmd,
    iVelOUT => Salidas.TR_P2_VF_Set,
    iRPM_a_HMI => HMI.StVeloc_TR_P2_VF); // Equipo_Motor_ATV320
HMI.StMarcha_TR_P2_VF := fbDosificador_P2.bEnMarcha;

// NETWORK 9
HMI.CmdM_TR_P2_VF R= HMI.bModo_Auto;

// NETWORK 10
Tmr_Alr_ZeroSpeed(IN := HMI.StMarcha_TR_P2_VF AND NOT entradas.TR_P2_ZS, PT := T#2s); // TON
hmi.TR_P2_Alr_ZS S= Tmr_Alr_ZeroSpeed.Q;

// NETWORK 11
_w1 := hmi.TR_P2_Alr_ZS_RstAlr;
hmi.TR_P2_Alr_ZS_RstAlr R= _w1;
hmi.TR_P2_Alr_ZS R= _w1;

// NETWORK 12
_w2 := HMI.bModo_Auto AND Polvos.InyectarPolvo[2];
IF _w2 THEN
    Tiempo_seg_to_TIME_TDemoraInyec(Segundos := REceta_activa.SetCircuitosPo[2].Demora, tTime => Auxtdemora); // Tiempo_seg_to_TIME
END_IF
TDemoraInyectarPolvo(IN := _w2, PT := Auxtdemora); // TON

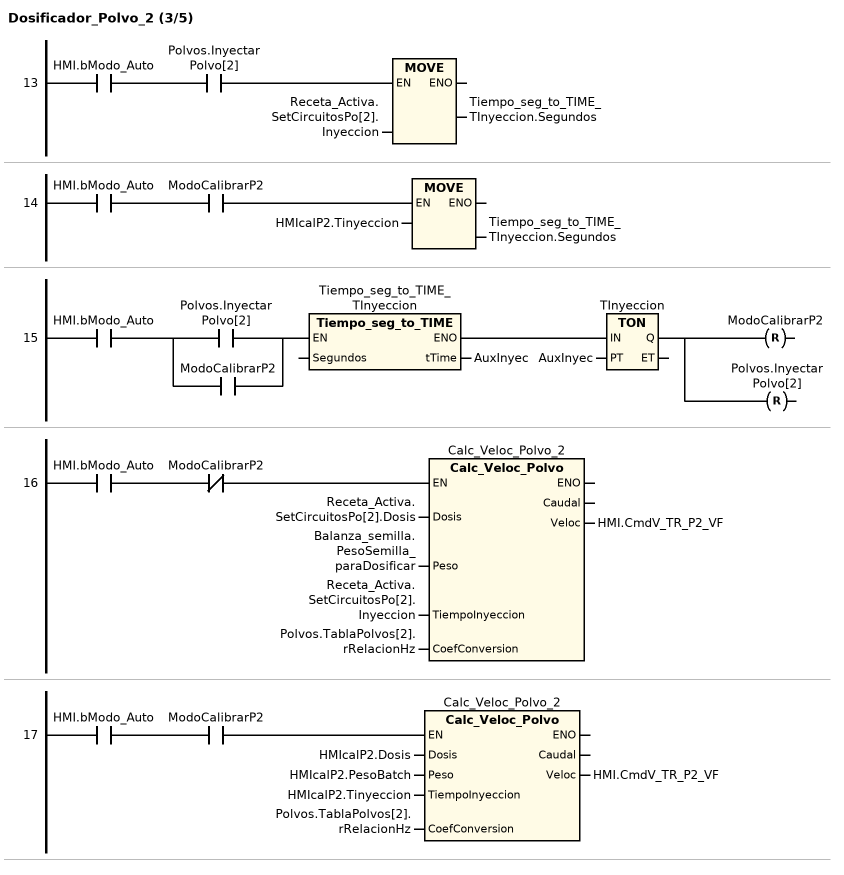
// NETWORK 13
IF HMI.bModo_Auto AND Polvos.InyectarPolvo[2] THEN
    Tiempo_seg_to_TIME_TInyeccion.Segundos := Receta_Activa.SetCircuitosPo[2].Inyeccion;
END_IF

// NETWORK 14
IF HMI.bModo_Auto AND ModoCalibrarP2 THEN Tiempo_seg_to_TIME_TInyeccion.Segundos := HMIcalP2.Tinyeccion; END_IF

// NETWORK 15
_w3 := HMI.bModo_Auto AND (Polvos.InyectarPolvo[2] OR ModoCalibrarP2);
IF _w3 THEN
    Tiempo_seg_to_TIME_TInyeccion(tTime => AuxInyec); // Tiempo_seg_to_TIME
END_IF
TInyeccion(IN := _w3, PT := AuxInyec); // TON
ModoCalibrarP2 R= TInyeccion.Q;
Polvos.InyectarPolvo[2] R= TInyeccion.Q;

// NETWORK 16
IF HMI.bModo_Auto AND NOT ModoCalibrarP2 THEN
    Calc_Veloc_Polvo_2(
        Dosis := Receta_Activa.SetCircuitosPo[2].Dosis,
        Peso := Balanza_semilla.PesoSemilla_paraDosificar,
        TiempoInyeccion := Receta_Activa.SetCircuitosPo[2].Inyeccion,
        CoefConversion := Polvos.TablaPolvos[2].rRelacionHz,
        Veloc => HMI.CmdV_TR_P2_VF); // Calc_Veloc_Polvo
END_IF

// NETWORK 17
IF HMI.bModo_Auto AND ModoCalibrarP2 THEN
    Calc_Veloc_Polvo_2(
        Dosis := HMIcalP2.Dosis,
        Peso := HMIcalP2.PesoBatch,
        TiempoInyeccion := HMIcalP2.Tinyeccion,
        CoefConversion := Polvos.TablaPolvos[2].rRelacionHz,
        Veloc => HMI.CmdV_TR_P2_VF); // Calc_Veloc_Polvo
END_IF

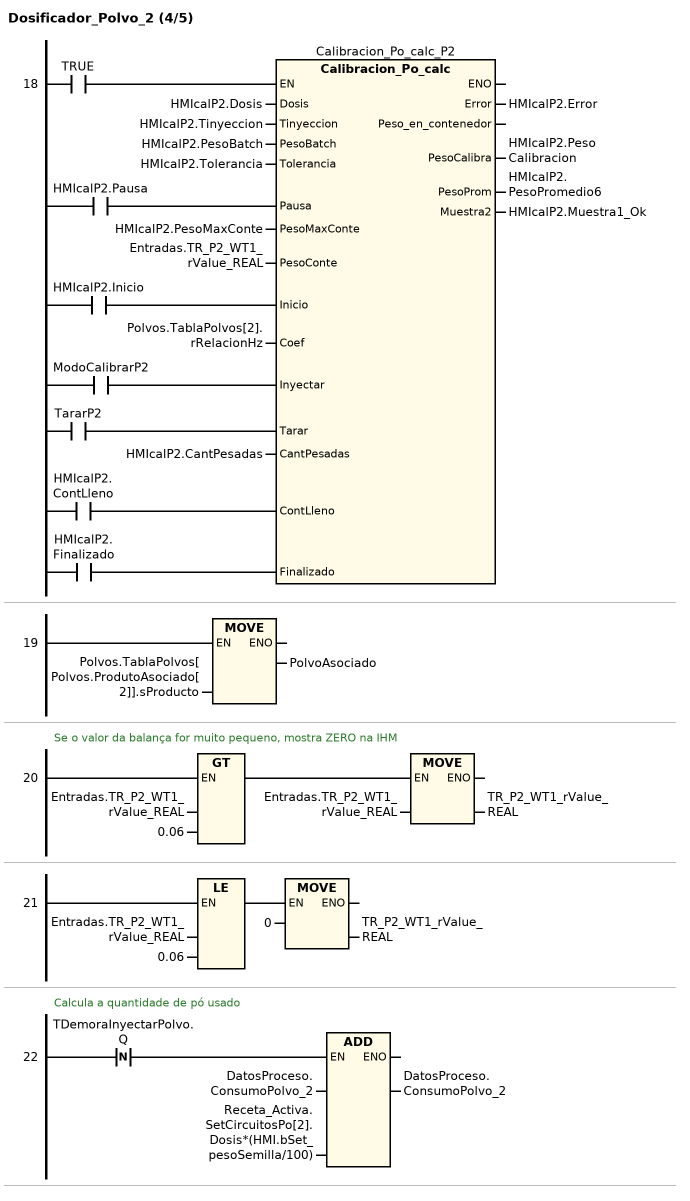
// NETWORK 18
Calibracion_Po_calc_P2(
    Dosis := HMIcalP2.Dosis,
    Tinyeccion := HMIcalP2.Tinyeccion,
    PesoBatch := HMIcalP2.PesoBatch,
    Tolerancia := HMIcalP2.Tolerancia,
    Pausa := HMIcalP2.Pausa,
    PesoMaxConte := HMIcalP2.PesoMaxConte,
    PesoConte := Entradas.TR_P2_WT1_rValue_REAL,
    Inicio := HMIcalP2.Inicio,
    Coef := Polvos.TablaPolvos[2].rRelacionHz,
    Inyectar := ModoCalibrarP2,
    Tarar := TararP2,
    CantPesadas := HMIcalP2.CantPesadas,
    ContLleno := HMIcalP2.ContLleno,
    Finalizado := HMIcalP2.Finalizado,
    Error => HMIcalP2.Error,
    PesoCalibra => HMIcalP2.PesoCalibracion,
    PesoProm => HMIcalP2.PesoPromedio6,
    Muestra2 => HMIcalP2.Muestra1_Ok); // Calibracion_Po_calc

// NETWORK 19
PolvoAsociado := Polvos.TablaPolvos[Polvos.ProdutoAsociado[2]].sProducto;

// NETWORK 20
// Se o valor da balança for muito pequeno, mostra ZERO na IHM
IF Entradas.TR_P2_WT1_rValue_REAL > 0.06 THEN TR_P2_WT1_rValue_REAL := Entradas.TR_P2_WT1_rValue_REAL; END_IF

// NETWORK 21
IF Entradas.TR_P2_WT1_rValue_REAL <= 0.06 THEN TR_P2_WT1_rValue_REAL := 0; END_IF

// NETWORK 22
// Calcula a quantidade de pó usado
_ft1(CLK := TDemoraInyectarPolvo.Q);
IF _ft1.Q THEN
    DatosProceso.ConsumoPolvo_2 := DatosProceso.ConsumoPolvo_2 + (Receta_Activa.SetCircuitosPo[2].Dosis*(HMI.bSet_pesoSemilla/100));
END_IF

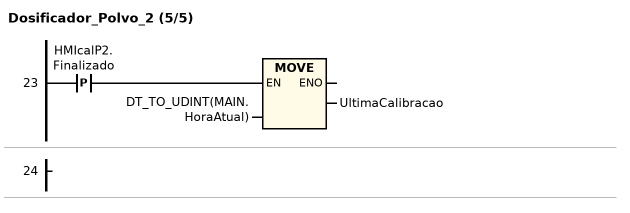
// NETWORK 23
_rt1(CLK := HMIcalP2.Finalizado);
IF _rt1.Q THEN UltimaCalibracao := DT_TO_UDINT(MAIN.HoraAtual); END_IF

// NETWORK 24

END_PROGRAM

// ---- POUs/Testes Thiago/IntervaloLavCalibr.TcPOU
PROGRAM IntervaloLavCalibr
VAR PERSISTENT
	IntervaloLavagem	:UDINT;	//Intervalo entre lavagens - Vem da IHM (h)
	AlarmeLavagem		:BOOL;	//Alguma linha excedeu o tempo de lavagem
	LinhaLavagem		:INT;	//Linha que excedeu o tempo de lavagem
	
	IntervaloCalibracao	:UDINT;	//Intervalo entre calibrações - Vem da IHM (h)
	AlarmeCalibracao	:BOOL;	//Alguma linha excedeu o tempo de calibração
	LinhaCalibracao		:INT;	//Linha que excedeu o tempo de calibração
	
END_VAR

VAR
	
	teste:LINT;
	teste2:LINT;
	TOF_Alarme: TOF;
	TOF_Calibracao: TOF;
END_VAR

//Essa rotina verifica se alguma calibração ou lavagem excedeu o tempo definido, subindo um alarme na IHM

//Verifica se alguma linha escedeu o intervalo entre lavagens. A primeira detectada, gera um alarme na IHM
TOF_Alarme(IN:= AlarmeLavagem, PT:= T#1S, Q=> , ET=> );	//Temporizador para garantir que a IHM conseguirá detectar a borda de subida do alarme
TOF_Calibracao(IN:= AlarmeCalibracao, PT:= T#1S, Q=> , ET=> );	//Temporizador para garantir que a IHM conseguirá detectar a borda de subida do alarme

{Region "Alarmes da lavagem}
	AlarmeLavagem := FALSE;	//Inicia a variável
	IF (DT_TO_LINT(Main.HoraAtual) - Liquidos.UltimoAlrLavagem[1]) > IntervaloLavagem * 3600 THEN
		Liquidos.UltimoAlrLavagem[1] := DT_TO_LINT(Main.HoraAtual) + (IntervaloLavagem * 360); 
		AlarmeLavagem := TRUE;
		LinhaLavagem := 1;
			
	ELSIF (DT_TO_LINT(Main.HoraAtual) - Liquidos.UltimoAlrLavagem[2]) > IntervaloLavagem * 3600 THEN
		Liquidos.UltimoAlrLavagem[2] := DT_TO_LINT(Main.HoraAtual) + (IntervaloLavagem * 360);
		AlarmeLavagem := TRUE;
		LinhaLavagem := 2;	
			
	ELSIF (DT_TO_LINT(Main.HoraAtual) - Liquidos.UltimoAlrLavagem[3]) > IntervaloLavagem * 3600 THEN
		Liquidos.UltimoAlrLavagem[3] := DT_TO_LINT(Main.HoraAtual) + (IntervaloLavagem * 360);
		AlarmeLavagem := TRUE;
		LinhaLavagem := 3;	
			
	ELSIF (DT_TO_LINT(Main.HoraAtual) - Liquidos.UltimoAlrLavagem[4]) > IntervaloLavagem * 3600 THEN
		Liquidos.UltimoAlrLavagem[4] := DT_TO_LINT(Main.HoraAtual) + (IntervaloLavagem * 360);
		AlarmeLavagem := TRUE;
		LinhaLavagem := 4;	
			
	ELSIF (DT_TO_LINT(Main.HoraAtual) - Liquidos.UltimoAlrLavagem[5]) > IntervaloLavagem * 3600 THEN
		Liquidos.UltimoAlrLavagem[5] := DT_TO_LINT(Main.HoraAtual) + (IntervaloLavagem * 360);
		AlarmeLavagem := TRUE;
		LinhaLavagem := 5;	
			
	ELSIF (DT_TO_LINT(Main.HoraAtual) - Liquidos.UltimoAlrLavagem[6]) > IntervaloLavagem * 3600 THEN
		Liquidos.UltimoAlrLavagem[6] := DT_TO_LINT(Main.HoraAtual) + (IntervaloLavagem * 360);
		AlarmeLavagem := TRUE;
		LinhaLavagem := 6;	
			
	ELSIF (DT_TO_UDINT(Main.HoraAtual) - Liquidos.UltimoAlrLavagem[7]) > IntervaloLavagem * 3600 THEN
		Liquidos.UltimoAlrLavagem[7] := DT_TO_LINT(Main.HoraAtual) + (IntervaloLavagem * 360);
		AlarmeLavagem := TRUE;
		LinhaLavagem := 7;	
			
	ELSIF (DT_TO_UDINT(Main.HoraAtual) - Liquidos.UltimoAlrLavagem[8]) > IntervaloLavagem * 3600 THEN
		Liquidos.UltimoAlrLavagem[8] := DT_TO_LINT(Main.HoraAtual) + (IntervaloLavagem * 360);
		AlarmeLavagem := TRUE;
		LinhaLavagem := 8;	
			
	ELSIF (DT_TO_LINT(Main.HoraAtual) - Liquidos.UltimoAlrLavagem[9]) > IntervaloLavagem * 3600 THEN
		Liquidos.UltimoAlrLavagem[9] := DT_TO_LINT(Main.HoraAtual) + (IntervaloLavagem * 360);
		AlarmeLavagem := TRUE;
		LinhaLavagem := 9;	
			
	ELSIF (DT_TO_LINT(Main.HoraAtual) - Liquidos.UltimoAlrLavagem[10]) > IntervaloLavagem * 3600 THEN
		Liquidos.UltimoAlrLavagem[10] := DT_TO_LINT(Main.HoraAtual) + (IntervaloLavagem * 360);
		AlarmeLavagem := TRUE;
		LinhaLavagem := 10;	
			
	ELSIF (DT_TO_LINT(Main.HoraAtual) - Liquidos.UltimoAlrLavagem[11]) > IntervaloLavagem * 3600 THEN
		Liquidos.UltimoAlrLavagem[11] := DT_TO_LINT(Main.HoraAtual) + (IntervaloLavagem * 360);
		AlarmeLavagem := TRUE;
		LinhaLavagem := 11;
				
	ELSIF (DT_TO_LINT(Main.HoraAtual) - Liquidos.UltimoAlrLavagem[12]) > IntervaloLavagem * 3600 THEN
		Liquidos.UltimoAlrLavagem[12] := DT_TO_LINT(Main.HoraAtual) + (IntervaloLavagem * 360);
		AlarmeLavagem := TRUE;
		LinhaLavagem := 12;
	END_IF
{endregion}

teste2 := DT_TO_LINT(Main.HoraAtual);
teste := (DT_TO_LINT(Main.HoraAtual) - HMI.UltimoAlrCalibr[1]);
{Region "Alarmes da calibração"}
	AlarmeCalibracao := FALSE;
	IF DT_TO_UDINT(Main.HoraAtual) - HMI.UltimoAlrCalibr[1] > IntervaloCalibracao * 3600 THEN
		HMI.UltimoAlrCalibr[1] := DT_TO_LINT(Main.HoraAtual) + (IntervaloCalibracao * 360);	//Se o alarme subir e a linha não for calibrada, o alarme subirá após 1/10 do intervalo
		AlarmeCalibracao := TRUE;
		LinhaCalibracao := 1;
	ELSIF DT_TO_UDINT(Main.HoraAtual) - HMI.UltimoAlrCalibr[2] > IntervaloCalibracao * 3600 THEN
		HMI.UltimoAlrCalibr[2] := DT_TO_LINT(Main.HoraAtual) + (IntervaloCalibracao * 360);	//Se o alarme subir e a linha não for calibrada, o alarme subirá após 1/10 do intervalo
		AlarmeCalibracao := TRUE;
		LinhaCalibracao := 2;
	ELSIF DT_TO_UDINT(Main.HoraAtual) - HMI.UltimoAlrCalibr[3] > IntervaloCalibracao * 3600 THEN
		HMI.UltimoAlrCalibr[3] := DT_TO_LINT(Main.HoraAtual) + (IntervaloCalibracao * 360);	//Se o alarme subir e a linha não for calibrada, o alarme subirá após 1/10 do intervalo
		AlarmeCalibracao := TRUE;
		LinhaCalibracao := 3;
	ELSIF DT_TO_UDINT(Main.HoraAtual) - HMI.UltimoAlrCalibr[4] > IntervaloCalibracao * 3600 THEN
		HMI.UltimoAlrCalibr[4] := DT_TO_LINT(Main.HoraAtual) + (IntervaloCalibracao * 360);	//Se o alarme subir e a linha não for calibrada, o alarme subirá após 1/10 do intervalo
		AlarmeCalibracao := TRUE;
		LinhaCalibracao := 4;
	ELSIF DT_TO_UDINT(Main.HoraAtual) - HMI.UltimoAlrCalibr[5] > IntervaloCalibracao * 3600 THEN
		HMI.UltimoAlrCalibr[5] := DT_TO_LINT(Main.HoraAtual) + (IntervaloCalibracao * 360);	//Se o alarme subir e a linha não for calibrada, o alarme subirá após 1/10 do intervalo
		AlarmeCalibracao := TRUE;
		LinhaCalibracao := 5;
	ELSIF DT_TO_UDINT(Main.HoraAtual) - HMI.UltimoAlrCalibr[6] > IntervaloCalibracao * 3600 THEN
		HMI.UltimoAlrCalibr[6] := DT_TO_LINT(Main.HoraAtual) + (IntervaloCalibracao * 360);	//Se o alarme subir e a linha não for calibrada, o alarme subirá após 1/10 do intervalo
		AlarmeCalibracao := TRUE;
		LinhaCalibracao := 6;
	ELSIF DT_TO_UDINT(Main.HoraAtual) - HMI.UltimoAlrCalibr[7] > IntervaloCalibracao * 3600 THEN
		HMI.UltimoAlrCalibr[7] := DT_TO_LINT(Main.HoraAtual) + (IntervaloCalibracao * 360);	//Se o alarme subir e a linha não for calibrada, o alarme subirá após 1/10 do intervalo
		AlarmeCalibracao := TRUE;
		LinhaCalibracao := 7;
	ELSIF DT_TO_UDINT(Main.HoraAtual) - HMI.UltimoAlrCalibr[8] > IntervaloCalibracao * 3600 THEN
		HMI.UltimoAlrCalibr[8] := DT_TO_LINT(Main.HoraAtual) + (IntervaloCalibracao * 360);	//Se o alarme subir e a linha não for calibrada, o alarme subirá após 1/10 do intervalo
		AlarmeCalibracao := TRUE;
		LinhaCalibracao := 8;
	ELSIF DT_TO_UDINT(Main.HoraAtual) - HMI.UltimoAlrCalibr[9] > IntervaloCalibracao * 3600 THEN
		HMI.UltimoAlrCalibr[9] := DT_TO_LINT(Main.HoraAtual) + (IntervaloCalibracao * 360);	//Se o alarme subir e a linha não for calibrada, o alarme subirá após 1/10 do intervalo
		AlarmeCalibracao := TRUE;
		LinhaCalibracao := 9;
	ELSIF DT_TO_UDINT(Main.HoraAtual) - HMI.UltimoAlrCalibr[10] > IntervaloCalibracao * 3600 THEN
		HMI.UltimoAlrCalibr[10] := DT_TO_LINT(Main.HoraAtual) + (IntervaloCalibracao * 360);	//Se o alarme subir e a linha não for calibrada, o alarme subirá após 1/10 do intervalo
		AlarmeCalibracao := TRUE;
		LinhaCalibracao := 10;
	ELSIF DT_TO_UDINT(Main.HoraAtual) - HMI.UltimoAlrCalibr[11] > IntervaloCalibracao * 3600 THEN
		HMI.UltimoAlrCalibr[11] := DT_TO_LINT(Main.HoraAtual) + (IntervaloCalibracao * 360);	//Se o alarme subir e a linha não for calibrada, o alarme subirá após 1/10 do intervalo
		AlarmeCalibracao := TRUE;
		LinhaCalibracao := 11;
	ELSIF DT_TO_UDINT(Main.HoraAtual) - HMI.UltimoAlrCalibr[12] > IntervaloCalibracao * 3600 THEN
		HMI.UltimoAlrCalibr[12] := DT_TO_LINT(Main.HoraAtual) + (IntervaloCalibracao * 360);	//Se o alarme subir e a linha não for calibrada, o alarme subirá após 1/10 do intervalo
		AlarmeCalibracao := TRUE;
		LinhaCalibracao := 12;
	END_IF
{endregion}

END_PROGRAM

// ---- POUs/Testes Thiago/iPC_Diagnostic.TcPOU
PROGRAM iPC_Diagnostic
VAR CONSTANT
	cNetId			: T_AmsNetID := '';				// local
END_VAR
VAR
	eState			: E_State := E_State.Init;
	
	//Informações do iPC
	sDeviceName		:STRING(39);	//Nome do dispositivo
	nTcBuild		:STRING;			//Versão do twincat
	CpuName			:STRING;		//Nome da CPU
	HardwareVersion	:STRING(100);		//Versão de hardware
	iPCSerialNumber	:STRING;		//Numero de série do IPC
	TCStatus		:UINT;		//Status do twincat
	
	//Desempenho do sistema
	nCpuFreq		:UDINT;			//Frequencia da CPU
	CpuTemp			:INT;			//Temperatura da CPU
	MB_Temperature	:INT;			//Temperatura da placa mãe
	MB_MaxTemperature	:DINT;			//Temperatura máximada placa mãe
	CpuUsage		:UINT;			//Uso da CPU
	OperationTime	:UDINT;			//Tempo de operação
	TotalMRAM		:ULINT;			//Memória ram total
	FreeMRAM		:ULINT;			//Memória ram em uso
	
	//Energia e armazenamento
	ulFreeDisk		:ULINT;			//Espaço livre no disco C
	ulTotalDisk		:ULINT;			//Espaço livre no disco C
	UPSBattCapacity	:USINT;			//Capacidade da bateria UPS
	UPSBattStatus	:USINT;		//Status da bateria UPS - 0-Unknown, 1-OK, 2-Change Battery
	
	//IPCDiag
	fbDiagRegister	: FB_IPCDiag_Register := (sNetId:=cNetId);
	
	//Leitura dos parâmetros
	
	//Informações do iPC
	fbDeviceName		: FB_IPCDiag_ReadParameterPeriodic := (eParameterKey:=E_IPCDiag_ParameterKey.IPCDeviceName, tPeriod:= T#10M, sNetId:=cNetId);
	fbTcBuild			: FB_IPCDiag_ReadParameterPeriodic := (eParameterKey:=E_IPCDiag_ParameterKey.TC_Version, tPeriod:= T#10M, sNetId:=cNetId);
	fbCpuName			: FB_IPCDiag_ReadParameterPeriodic := (eParameterKey:=E_IPCDiag_ParameterKey.CPU_Name, tPeriod:= T#10M, sNetId:=cNetId);
	fbHWVersion			: FB_IPCDiag_ReadParameterPeriodic := (eParameterKey:=E_IPCDiag_ParameterKey.IPCHardwareVersion, tPeriod:= T#10M, sNetId:=cNetId);
	fbiPCSerialNumber	: FB_IPCDiag_ReadParameterPeriodic := (eParameterKey:=E_IPCDiag_ParameterKey.IPCSerialNumber, tPeriod:= T#10M, sNetId:=cNetId);
	fbTCStatus			: FB_IPCDiag_ReadParameterPeriodic := (eParameterKey:=E_IPCDiag_ParameterKey.TC_Status, tPeriod:= T#10S, sNetId:=cNetId);
	
	//Desempenho do sistema
	fbCpuFreq			: FB_IPCDiag_ReadParameterPeriodic := (eParameterKey:=E_IPCDiag_ParameterKey.CPU_Frequency, tPeriod:= T#2S, sNetId:=cNetId);
	fbCpuTemp			: FB_IPCDiag_ReadParameterPeriodic := (eParameterKey:=E_IPCDiag_ParameterKey.CPU_Temp, tPeriod:= T#2S, sNetId:=cNetId);
	fbMBTemp			: FB_IPCDiag_ReadParameterPeriodic := (eParameterKey:=E_IPCDiag_ParameterKey.MB_Temperature, tPeriod:= T#2S, sNetId:=cNetId);
	fbMBMaxTemp			: FB_IPCDiag_ReadParameterPeriodic := (eParameterKey:=E_IPCDiag_ParameterKey.MB_MaxTemperature, tPeriod:= T#60S, sNetId:=cNetId);
	fbCpuUsage			: FB_IPCDiag_ReadParameterPeriodic := (eParameterKey:=E_IPCDiag_ParameterKey.CPU_Usage, tPeriod:= T#2S, sNetId:=cNetId);
	fbOpTime			: FB_IPCDiag_ReadParameterPeriodic := (eParameterKey:=E_IPCDiag_ParameterKey.MB_OperationTime, tPeriod:= T#3M, sNetId:=cNetId);
	fbTotalMRam			: FB_IPCDiag_ReadParameterPeriodic := (eParameterKey:=E_IPCDiag_ParameterKey.Memory_ProgramMemoryAllocated, tPeriod:= T#3M, sNetId:=cNetId);
	fbFreeMRam			: FB_IPCDiag_ReadParameterPeriodic := (eParameterKey:=E_IPCDiag_ParameterKey.Memory_ProgramMemoryAvailable, tPeriod:= T#2S, sNetId:=cNetId);
	
	//Energia e armazenamento
	fbFreeDisk			: FB_IPCDiag_ReadParameterPeriodic := (eParameterKey:=E_IPCDiag_ParameterKey.Disk_FreeSpaceOfVolumeC, tPeriod:= T#10S, sNetId:=cNetId);
	fbTotalSize		: FB_IPCDiag_ReadParameterPeriodic := (eParameterKey:=E_IPCDiag_ParameterKey.Disk_VolumeList_TotelSize, tPeriod:= T#1M, sNetId:=cNetId);
	fbUPSCap			: FB_IPCDiag_ReadParameterPeriodic := (eParameterKey:=E_IPCDiag_ParameterKey.UPS_BatteryCapacity, tPeriod:= T#10S, sNetId:=cNetId);
	fbUPSStatus			: FB_IPCDiag_ReadParameterPeriodic := (eParameterKey:=E_IPCDiag_ParameterKey.UPS_BatteryStatus, tPeriod:= T#10S, sNetId:=cNetId);
	
	//Ajuste dos valores de memória
	rFreeRAM:REAL;
	rTotalRAM:REAL;
	rFreeDisk:REAL;
	rDiskTotalSize:REAL;;
END_VAR

//Esse programa faz a leitura dos parâmetros do iPC

CASE eState OF
E_State.Init:
	IF NOT fbDiagRegister.bBusy THEN
		fbDiagRegister(bExecute:=TRUE); // need to be executed once
	ELSE
		fbDiagRegister(bExecute:=FALSE);
	END_IF
	IF NOT fbDiagRegister.bBusy THEN
		IF fbDiagRegister.bError THEN
			eState := E_State.Error;
		ELSE
			eState := E_State.Idle;
		END_IF
	END_IF
E_State.Idle:
		eState := E_State.ReadPeriodically;
		
E_State.ReadPeriodically:

	{Region "Informações do iPC"}	//Informações do iPC
		//Nome do dispositivo
		fbDeviceName(bEnable:=TRUE, fbRegister:=fbDiagRegister);
		IF fbDeviceName.bValid THEN
			fbDeviceName.GetParameter(pBuffer:=ADR(sDeviceName), nBufferSize:=SIZEOF(sDeviceName) );	
		END_IF
		
		//Versão do twincat
		fbTcBuild(bEnable:=TRUE, fbRegister:=fbDiagRegister);
		IF fbTcBuild.bValid THEN
			fbTcBuild.GetParameter(pBuffer:=ADR(nTcBuild), nBufferSize:=SIZEOF(nTcBuild) );	
		END_IF
		
		//Nome da CPU
		fbCpuName(bEnable:=TRUE, fbRegister:=fbDiagRegister);
		IF fbCpuName.bValid THEN
			fbCpuName.GetParameter(pBuffer:=ADR(CpuName), nBufferSize:=SIZEOF(CpuName) );
		END_IF
		
		//Versão do hardware
		fbHWVersion(bEnable:=TRUE, fbRegister:=fbDiagRegister);
		IF fbHWVersion.bValid THEN
			fbHWVersion.GetParameter(pBuffer:=ADR(HardwareVersion), nBufferSize:=SIZEOF(HardwareVersion) );	
		END_IF
		
		//Numero de série do iPC
		fbiPCSerialNumber(bEnable:=TRUE, fbRegister:=fbDiagRegister);
		IF fbiPCSerialNumber.bValid THEN
			fbiPCSerialNumber.GetParameter(pBuffer:=ADR(iPCSerialNumber), nBufferSize:=SIZEOF(iPCSerialNumber) );	
		END_IF
		
		//Status do Twincat
		fbTCStatus(bEnable:=TRUE, fbRegister:=fbDiagRegister);
		IF fbTCStatus.bValid THEN
			fbTCStatus.GetParameter(pBuffer:=ADR(TCStatus), nBufferSize:=SIZEOF(TCStatus) );	
		END_IF
	{endregion}
	
	{Region "Desempenho do sistema"}
		//Frequencia do CPU
		fbCpuFreq(bEnable:=TRUE, fbRegister:=fbDiagRegister);
		IF fbCpuFreq.bValid THEN
			fbCpuFreq.GetParameter(pBuffer:=ADR(nCpuFreq), nBufferSize:=SIZEOF(nCpuFreq) );	
		END_IF
		//Temperatura do CPU
		fbCpuTemp(bEnable:=TRUE, fbRegister:=fbDiagRegister);
		IF fbCpuTemp.bValid THEN
			fbCpuTemp.GetParameter(pBuffer:=ADR(CpuTemp), nBufferSize:=SIZEOF(CpuTemp) );	
		END_IF
		//Temperatura da placa mae
		fbMBTemp(bEnable:=TRUE, fbRegister:=fbDiagRegister);
		IF fbMBTemp.bValid THEN
			fbMBTemp.GetParameter(pBuffer:=ADR(MB_Temperature), nBufferSize:=SIZEOF(MB_Temperature) );	
		END_IF
		//Temperatura máxima da placa mae
		fbMBMaxTemp(bEnable:=TRUE, fbRegister:=fbDiagRegister);
		IF fbMBMaxTemp.bValid THEN
			fbMBMaxTemp.GetParameter(pBuffer:=ADR(MB_MaxTemperature), nBufferSize:=SIZEOF(MB_MaxTemperature) );	
		END_IF
		//Uso do CPU
		fbCpuUsage(bEnable:=TRUE, fbRegister:=fbDiagRegister);
		IF fbCpuUsage.bValid THEN
			fbCpuUsage.GetParameter(pBuffer:=ADR(CpuUsage), nBufferSize:=SIZEOF(CpuUsage) );	
		END_IF
		//Tempo de operação
		fbOpTime(bEnable:=TRUE, fbRegister:=fbDiagRegister);
		IF fbOpTime.bValid THEN
			fbOpTime.GetParameter(pBuffer:=ADR(OperationTime), nBufferSize:=SIZEOF(OperationTime) );	
		END_IF
		//Total de RAM
		fbTotalMRam(bEnable:=TRUE, fbRegister:=fbDiagRegister);
		IF fbTotalMRam.bValid THEN
			fbTotalMRam.GetParameter(pBuffer:=ADR(TotalMRAM), nBufferSize:=SIZEOF(TotalMRAM) );	
			rTotalRAM := TO_REAL(TotalMRAM)/(1024*1024*1024);
		END_IF
		//RAM disponível
		fbFreeMRam(bEnable:=TRUE, fbRegister:=fbDiagRegister);
		IF fbFreeMRam.bValid THEN
			fbFreeMRam.GetParameter(pBuffer:=ADR(FreeMRAM), nBufferSize:=SIZEOF(FreeMRAM) );	
			rFreeRAM := TO_REAL(FreeMRAM)/(1024*1024*1024);
		END_IF
	{endregion}
	
	{Region "Energia e armazenamento"}		//Energia e armazenamento
	
		//Memória livre
		fbFreeDisk(bEnable:=TRUE, fbRegister:=fbDiagRegister);
		IF fbFreeDisk.bValid THEN
			fbFreeDisk.GetParameter(pBuffer:=ADR(ulFreeDisk), nBufferSize:=SIZEOF(ulFreeDisk) );	
			rFreeDisk := TO_REAL(ulFreeDisk)/(1024*1024*1024);
		END_IF
		//Memória total
		fbTotalSize(bEnable:=TRUE, fbRegister:=fbDiagRegister);
		IF fbTotalSize.bValid THEN
			fbTotalSize.GetParameter(pBuffer:=ADR(ulTotalDisk), nBufferSize:=SIZEOF(ulTotalDisk) );	
			rDiskTotalSize := TO_REAL(ulTotalDisk)/(1024*1024*1024);
		END_IF
		//Capacidade da bateria UPS
		fbUPSCap(bEnable:=TRUE, fbRegister:=fbDiagRegister);
		IF fbUPSCap.bValid THEN
			fbUPSCap.GetParameter(pBuffer:=ADR(UPSBattCapacity), nBufferSize:=SIZEOF(UPSBattCapacity) );	
		END_IF
		//Status da bateria UPS
		fbUPSStatus(bEnable:=TRUE, fbRegister:=fbDiagRegister);
		IF fbUPSStatus.bValid THEN
			fbUPSStatus.GetParameter(pBuffer:=ADR(UPSBattStatus), nBufferSize:=SIZEOF(UPSBattStatus) );	
		END_IF
	{endregion}
	
	
	

	
E_State.Error:
	(* implementation of error logging and error handling *)
	(* hint: An error could also occur if a parameter is not supported by chosen hardware or image. 
	E.g. not all IPCs offer a CPU temperature measurement. *)

END_CASE

END_PROGRAM

// ---- POUs/PasosDosificar.TcPOU
PROGRAM PasosDosificar
VAR_IN_OUT
	iStep:INT;
END_VAR
VAR
	counter:INT;
	dosificando1:BOOL;
	FinDosificado:BOOL;
END_VAR

//Antes de verificar a dosagem, desliga todas as bombas. É preciso para que não fique nenhuma bomba ligada caso o processo pare no meio	
(*FOR counter := 1 TO 12 DO
	Liquidos.InyectarLiq[counter]:=FALSE;
END_FOR
FOR counter := 1 TO 2 DO
	Polvos.InyectarPolvo[counter]:=TRUE	;
END_FOR
*)
CASE iStep OF
	1: counter:=1;
	IF NOT dosificando1 THEN
		FOR counter:=1 TO 12 BY 1 DO
			IF Receta_Activa.SetCircuitosLiq[counter].Paso=iStep THEN
				Liquidos.InyectarLiq[counter]:=TRUE	;
			END_IF
		END_FOR	
		FOR counter:=1 TO 2 BY 1 DO
			IF Receta_Activa.SetCircuitosPo[counter].Paso=iStep THEN
				Polvos.InyectarPolvo[counter]:=TRUE	;
			END_IF
		END_FOR		
	END_IF
	dosificando1:=Liquidos.InyectarLiq[1] OR Liquidos.InyectarLiq[2] OR Liquidos.InyectarLiq[3] OR Liquidos.InyectarLiq[4]OR Liquidos.InyectarLiq[5] OR Liquidos.InyectarLiq[6] OR Liquidos.InyectarLiq[7] OR Liquidos.InyectarLiq[8]OR Liquidos.InyectarLiq[9] OR Liquidos.InyectarLiq[10] OR Liquidos.InyectarLiq[11] OR Liquidos.InyectarLiq[12]OR Polvos.InyectarPolvo[1]OR Polvos.InyectarPolvo[2];
	IF NOT dosificando1 THEN
		iStep:=iStep+1;
	END_IF
	2: counter:=1;
	IF NOT dosificando1 THEN
	FOR counter:=1 TO 12 BY 1 DO
		IF Receta_Activa.SetCircuitosLiq[counter].Paso=iStep THEN
		Liquidos.InyectarLiq[counter]:=TRUE	;
		END_IF
	END_FOR	
	FOR counter:=1 TO 2 BY 1 DO
		IF Receta_Activa.SetCircuitosPo[counter].Paso=iStep THEN
		Polvos.InyectarPolvo[counter]:=TRUE	;
		END_IF
	END_FOR		
	END_IF
	dosificando1:=Liquidos.InyectarLiq[1] OR Liquidos.InyectarLiq[2] OR Liquidos.InyectarLiq[3] OR Liquidos.InyectarLiq[4]OR Liquidos.InyectarLiq[5] OR Liquidos.InyectarLiq[6] OR Liquidos.InyectarLiq[7] OR Liquidos.InyectarLiq[8]OR Liquidos.InyectarLiq[9] OR Liquidos.InyectarLiq[10] OR Liquidos.InyectarLiq[11] OR Liquidos.InyectarLiq[12]OR Polvos.InyectarPolvo[1]OR Polvos.InyectarPolvo[2];
	IF NOT dosificando1 THEN
		iStep:=iStep+1;
	END_IF
	3: counter:=1;
	IF NOT dosificando1 THEN
	FOR counter:=1 TO 12 BY 1 DO
		IF Receta_Activa.SetCircuitosLiq[counter].Paso=iStep THEN
		Liquidos.InyectarLiq[counter]:=TRUE	;
		END_IF
	END_FOR
	FOR counter:=1 TO 2 BY 1 DO
		IF Receta_Activa.SetCircuitosPo[counter].Paso=iStep THEN
		Polvos.InyectarPolvo[counter]:=TRUE	;
		END_IF
	END_FOR			
	END_IF
	dosificando1:=Liquidos.InyectarLiq[1] OR Liquidos.InyectarLiq[2] OR Liquidos.InyectarLiq[3] OR Liquidos.InyectarLiq[4]OR Liquidos.InyectarLiq[5] OR Liquidos.InyectarLiq[6] OR Liquidos.InyectarLiq[7] OR Liquidos.InyectarLiq[8]OR Liquidos.InyectarLiq[9] OR Liquidos.InyectarLiq[10] OR Liquidos.InyectarLiq[11] OR Liquidos.InyectarLiq[12]OR Polvos.InyectarPolvo[1]OR Polvos.InyectarPolvo[2];
	IF NOT dosificando1 THEN
		iStep:=iStep+1;
	END_IF
	4: counter:=1;
	IF NOT dosificando1 THEN
	FOR counter:=1 TO 12 BY 1 DO
		IF Receta_Activa.SetCircuitosLiq[counter].Paso=iStep THEN
		Liquidos.InyectarLiq[counter]:=TRUE	;
		END_IF
	END_FOR
	FOR counter:=1 TO 2 BY 1 DO
		IF Receta_Activa.SetCircuitosPo[counter].Paso=iStep THEN
		Polvos.InyectarPolvo[counter]:=TRUE	;
		END_IF
	END_FOR			
	END_IF
	dosificando1:=Liquidos.InyectarLiq[1] OR Liquidos.InyectarLiq[2] OR Liquidos.InyectarLiq[3] OR Liquidos.InyectarLiq[4]OR Liquidos.InyectarLiq[5] OR Liquidos.InyectarLiq[6] OR Liquidos.InyectarLiq[7] OR Liquidos.InyectarLiq[8]OR Liquidos.InyectarLiq[9] OR Liquidos.InyectarLiq[10] OR Liquidos.InyectarLiq[11] OR Liquidos.InyectarLiq[12]OR Polvos.InyectarPolvo[1]OR Polvos.InyectarPolvo[2];
	IF NOT dosificando1 THEN
		iStep:=iStep+1;
	END_IF
	5: counter:=1;
	IF NOT dosificando1 THEN
	FOR counter:=1 TO 12 BY 1 DO
		IF Receta_Activa.SetCircuitosLiq[counter].Paso=iStep THEN
		Liquidos.InyectarLiq[counter]:=TRUE	;
		END_IF
	END_FOR
	FOR counter:=1 TO 2 BY 1 DO
		IF Receta_Activa.SetCircuitosPo[counter].Paso=iStep THEN
		Polvos.InyectarPolvo[counter]:=TRUE	;
		END_IF
	END_FOR			
	END_IF
	dosificando1:=Liquidos.InyectarLiq[1] OR Liquidos.InyectarLiq[2] OR Liquidos.InyectarLiq[3] OR Liquidos.InyectarLiq[4]OR Liquidos.InyectarLiq[5] OR Liquidos.InyectarLiq[6] OR Liquidos.InyectarLiq[7] OR Liquidos.InyectarLiq[8]OR Liquidos.InyectarLiq[9] OR Liquidos.InyectarLiq[10] OR Liquidos.InyectarLiq[11] OR Liquidos.InyectarLiq[12]OR Polvos.InyectarPolvo[1]OR Polvos.InyectarPolvo[2];
	IF NOT dosificando1 THEN
		iStep:=iStep+1;
	END_IF
	6: counter:=1;
	IF NOT dosificando1 THEN
	FOR counter:=1 TO 12 BY 1 DO
		IF Receta_Activa.SetCircuitosLiq[counter].Paso=iStep THEN
		Liquidos.InyectarLiq[counter]:=TRUE	;
		END_IF
	END_FOR
	FOR counter:=1 TO 2 BY 1 DO
		IF Receta_Activa.SetCircuitosPo[counter].Paso=iStep THEN
		Polvos.InyectarPolvo[counter]:=TRUE	;
		END_IF
	END_FOR			
	END_IF
	dosificando1:=Liquidos.InyectarLiq[1] OR Liquidos.InyectarLiq[2] OR Liquidos.InyectarLiq[3] OR Liquidos.InyectarLiq[4]OR Liquidos.InyectarLiq[5] OR Liquidos.InyectarLiq[6] OR Liquidos.InyectarLiq[7] OR Liquidos.InyectarLiq[8]OR Liquidos.InyectarLiq[9] OR Liquidos.InyectarLiq[10] OR Liquidos.InyectarLiq[11] OR Liquidos.InyectarLiq[12]OR Polvos.InyectarPolvo[1]OR Polvos.InyectarPolvo[2];
	IF NOT dosificando1 THEN
		iStep:=iStep+1;
	END_IF
	7: counter:=1;
	IF NOT dosificando1 THEN
	FOR counter:=1 TO 12 BY 1 DO
		IF Receta_Activa.SetCircuitosLiq[counter].Paso=iStep THEN
		Liquidos.InyectarLiq[counter]:=TRUE	;
		END_IF
	END_FOR
	FOR counter:=1 TO 2 BY 1 DO
		IF Receta_Activa.SetCircuitosPo[counter].Paso=iStep THEN
		Polvos.InyectarPolvo[counter]:=TRUE	;
		END_IF
	END_FOR			
	END_IF
	dosificando1:=Liquidos.InyectarLiq[1] OR Liquidos.InyectarLiq[2] OR Liquidos.InyectarLiq[3] OR Liquidos.InyectarLiq[4]OR Liquidos.InyectarLiq[5] OR Liquidos.InyectarLiq[6] OR Liquidos.InyectarLiq[7] OR Liquidos.InyectarLiq[8]OR Liquidos.InyectarLiq[9] OR Liquidos.InyectarLiq[10] OR Liquidos.InyectarLiq[11] OR Liquidos.InyectarLiq[12]OR Polvos.InyectarPolvo[1]OR Polvos.InyectarPolvo[2];
	IF NOT dosificando1 THEN
		iStep:=iStep+1;
	END_IF
	8: counter:=1;
	IF NOT dosificando1 THEN
		FOR counter:=1 TO 12 BY 1 DO
			IF Receta_Activa.SetCircuitosLiq[counter].Paso=iStep THEN
			Liquidos.InyectarLiq[counter]:=TRUE	;
			END_IF
		END_FOR
		FOR counter:=1 TO 2 BY 1 DO
			IF Receta_Activa.SetCircuitosPo[counter].Paso=iStep THEN
			Polvos.InyectarPolvo[counter]:=TRUE	;
			END_IF
		END_FOR			
	END_IF
	dosificando1:=Liquidos.InyectarLiq[1] OR Liquidos.InyectarLiq[2] OR Liquidos.InyectarLiq[3] OR Liquidos.InyectarLiq[4]OR Liquidos.InyectarLiq[5] OR Liquidos.InyectarLiq[6] OR Liquidos.InyectarLiq[7] OR Liquidos.InyectarLiq[8]OR Liquidos.InyectarLiq[9] OR Liquidos.InyectarLiq[10] OR Liquidos.InyectarLiq[11] OR Liquidos.InyectarLiq[12]OR Polvos.InyectarPolvo[1]OR Polvos.InyectarPolvo[2];
	IF NOT dosificando1 THEN
		iStep:=iStep+1;
	END_IF
	ELSE
		FinDosificado:=TRUE;
END_CASE

END_PROGRAM

// ---- POUs/_Seguridad.TcPOU
PROGRAM _Seguridad
VAR
END_VAR

Seguridad.Run := TRUE;
Seguridad.Restart		:= Entradas.ReposicionEmerg OR HMI.Restart;
Seguridad.ErrorAck		:= Entradas.ReposicionEmerg OR HMI.Restart;
Seguridad.ResetPorta	:= Entradas.ReposicionEmerg OR HMI.Restart;

IF HMI.Restart THEN
	HMI.Restart := FALSE;
END_IF

IF NOT Seguridad.PB_Emergencia THEN
	Liquidos.InyectarLiq[1] := FALSE;
	Liquidos.InyectarLiq[2] := FALSE;
	Liquidos.InyectarLiq[3] := FALSE;
	Liquidos.InyectarLiq[4] := FALSE;
	Liquidos.InyectarLiq[5] := FALSE;
	Liquidos.InyectarLiq[6] := FALSE;
	Liquidos.InyectarLiq[7] := FALSE;
	Liquidos.InyectarLiq[8] := FALSE; //a
	Liquidos.InyectarLiq[9] := FALSE;
	Liquidos.InyectarLiq[10] := FALSE;
	Liquidos.InyectarLiq[11] := FALSE;
	Liquidos.InyectarLiq[12] := FALSE;
	Polvos.InyectarPolvo[1] := FALSE;
	Polvos.InyectarPolvo[2] := FALSE;
END_IF

END_PROGRAM

// ---- POUs/Alarmas.TcPOU
PROGRAM Alarmas
VAR
	Resumen_alarmas_BombasLiquidos:BOOL;
	Alarmas_agitadores:INT;
	AL_verde :BOOL;
	AL_verde_fija :BOOL;
	Al_azul	 :BOOL;
	AL_roja  :BOOL;
	AL_amarilla:BOOL;
	AL_nula  :BOOL;
	Ac_aviso :BOOL;
	Ac_alarma:BOOL;
	Ac_nula :BOOL;
	
	Ac_AlarmePorta: BOOL;
	
	// Mapeamento de alarmes da máquina
	AlarmesMaquina: INT;
END_VAR

Resumen_alarmas_BombasLiquidos :=	HMI.PP1_L1_AG_Alr OR 
									HMI.PP1_L2_AG_Alr OR 
									HMI.PP1_L3_AG_Alr OR 
									HMI.PP1_L4_AG_Alr OR 
									HMI.PP2_L5_AG_Alr OR 
									HMI.PP2_L6_AG_Alr OR 
									HMI.PP2_L7_AG_Alr OR  
									HMI.PP2_L8_AG_Alr OR  
									HMI.PP3_L9_AG_Alr OR  
									HMI.PP3_L10_AG_Alr OR  
									HMI.PP3_L11_AG_Alr OR  
									HMI.PP3_L12_AG_Alr;
Alarmas_agitadores.0:=HMI.PP1_L1_AG_Alr;
Alarmas_agitadores.1:=HMI.PP1_L2_AG_Alr;
Alarmas_agitadores.2:=HMI.PP1_L3_AG_Alr;

AL_verde_fija	:= seguridad.PB_Emergencia AND HMI.bRun;
AL_verde		:= INICIO.Premarcha;	
AL_azul			:= seguridad.PB_Emergencia AND NOT HMI.bRun;
AL_roja			:= NOT seguridad.PB_Emergencia;
AL_nula			:= NOT AL_verde AND NOT AL_roja AND NOT AL_azul;
Ac_Aviso		:= INICIO.Premarcha;
Ac_alarma		:= Resumen_alarmas_BombasLiquidos;
AC_nula			:= NOT Ac_Aviso AND NOT Ac_alarma;
Ac_AlarmePorta	:= NOT Seguridad.ParadaDePorta;

//Rodando
IF AL_verde_fija THEN
	Salidas.TR_AL2_L:=2;	
END_IF

//Máquina OK, sem produzir
IF AL_azul THEN
	Salidas.TR_AL2_L:=4;	
END_IF

//Em pré marcha
IF AL_verde THEN
	Salidas.TR_AL2_L:=50;
END_IF

//Desliga led
IF AL_nula THEN
	Salidas.TR_AL2_L:=0;
END_IF

//Parada de porta
IF Ac_AlarmePorta THEN
	Salidas.TR_AL2_L := 56;
END_IF

//Em emergência
IF AL_roja THEN
	Salidas.TR_AL2_L:=49;
END_IF

Salidas.TR_AL1_L:=Salidas.TR_AL2_L;

IF Ac_Aviso THEN
	Salidas.TR_AL2_Ac:=81;
END_IF

IF Ac_nula THEN
	Salidas.TR_AL2_Ac:=0;
END_IF

IF Alarmas_agitadores<>0 THEN 
	Salidas.TR_AL1_L:=17;
END_IF


AlarmesMaquina := 0;	//Tudo OK. Começa em zero. Se tiver algum alarme, o valor do mapeamento é atribuido abaixo
//Mapeamento de alarmes para alterar o texto no rodapé da IHM
IF NOT Seguridad.PB_Emergencia THEN
	AlarmesMaquina := 1;	//Em emergência
ELSIF NOT Entradas.TR_S_PDI THEN
	AlarmesMaquina := 2;	//Sem pressão pneumática
ELSIF NOT SafetyInputs.TR2_E1_CH01 OR NOT SafetyInputs.TR2_E1_CH02 THEN
	AlarmesMaquina := 3;	//Tampa frontal da balança
ELSIF NOT SafetyInputs.TR2_E2_CH01 OR NOT SafetyInputs.TR2_E2_CH02 THEN
	AlarmesMaquina := 4;	//Tampa traseira da balança
ELSIF NOT SafetyInputs.TR2_E3_CH01 OR NOT SafetyInputs.TR2_E3_CH02 THEN
	AlarmesMaquina := 5;	//Tampa esquerda da balança
ELSIF NOT SafetyInputs.TR2_E4_CH01 OR NOT SafetyInputs.TR2_E4_CH02 THEN
	AlarmesMaquina := 6;	//Tampa direita da balança
ELSIF NOT SafetyInputs.TR3_E1_CH01 OR NOT SafetyInputs.TR3_E1_CH02 THEN
	AlarmesMaquina := 7;	//Tampa frontal inferior da balança
ELSIF NOT SafetyInputs.TR3_E2_CH01 OR NOT SafetyInputs.TR3_E2_CH02 THEN
	AlarmesMaquina := 8;	//Tampa traSeira inferior da balança
ELSIF NOT SafetyInputs.TR3_E3_CH01 OR NOT SafetyInputs.TR3_E3_CH02 THEN
	AlarmesMaquina := 9;	//Tampas do homogeneizador
ELSIF NOT SafetyInputs.TR3_E4_CH01 OR NOT SafetyInputs.TR3_E4_CH02 THEN
	AlarmesMaquina := 10;	//Tampa da porta de inspeção da balança
ELSIF NOT Seguridad.ParadaDePorta THEN
	AlarmesMaquina := 11;	//Parada de porta. Falta RESET
ELSIF HMI.bModo_Auto THEN
	IF Tratadora.fbHomogenizador.wEstado = 0 THEN
		AlarmesMaquina := 12;	//Inversor do homogeneizador desligado
	ELSIF Tratadora.fbAspersor.wEstado = 0 THEN
		AlarmesMaquina := 13;	//Inversor do aspersor desligado
	END_IF;
ELSIF HMI.bRun AND (Receta_activa.SetCircuitosPo[1].Paso > 0 AND (NOT Entradas.TR_P1_ZC OR NOT entradas.TR_P1_LLS)) THEN
	AlarmesMaquina := 14;	//Pó 1 com nivel baixo ou fora de posição
ELSIF HMI.bRun AND (Receta_activa.SetCircuitosPo[2].Paso > 0 AND (NOT Entradas.TR_P2_ZC OR NOT entradas.TR_P2_LLS)) THEN
	AlarmesMaquina := 15;	//Pó 2 com nivel baixo ou fora de posição
ELSIF NOT Entradas.TR_S_LLS AND HMI.bRun THEN
	AlarmesMaquina := 16;	//Caixa superior sem sementes
ELSIF HMI.bRun AND Entradas.PE_B1_V1_ZO AND Entradas.PE_B2_V1_ZO AND Entradas.PE_B3_V1_ZO THEN
	AlarmesMaquina := 17;	//Nenhuma descarga das caixas de ensaque está ativa
ELSIF Resumen_alarmas_BombasLiquidos THEN
	AlarmesMaquina := 18;	//Falha nos agitadores
ELSIF (HMI.bModo_Pausa OR Descarga_Semilla.PausaEnsaque) AND HMI.bModo_Auto THEN
	AlarmesMaquina := 19;	//Máquina pausada
ELSE
	AlarmesMaquina := 0;	//Tudo OK
END_IF

END_PROGRAM

// ---- POUs/Testes Thiago/PRG_DE_TESTES.TcPOU
PROGRAM PRG_DE_TESTES
VAR
	Lavagem:Lavagem;
	Calibracao: Calibracao_V02;
	FB_DBRead_0: FB_DBRead;
	grupo:STRING;
	hora:TIME;
	data:DATE;
	nome:STRING;
	mensagem:LREAL;
	EventLog:DINT;
	FB_DBConnectionAdd_0: FB_DBConnectionAdd;
	FB_DBCyclicRdWrt_0: FB_DBCyclicRdWrt;
	FB_DBConnectionAdd_1: FB_DBConnectionAdd;
	TesteAlarmes : ARRAY [1..3 ] OF GeraAlarme;
	AcionaEvento: BOOL;
	Confirma: BOOL;
	MediaMovel_0: MediaMovel;
	TON_teste: TON;
	SDO_READ_0: SDO_READ;
	FB_EcCoESdoRead_0: FB_EcCoESdoRead;
	SDO_READ_1: SDO_READ;
	Calibracao_V03_0: Calibracao_V03;
	DiagInfo:STRING;
	TesteApex:INT;
	FB_IPCDiag_ReadParameter_0: FB_IPCDiag_ReadParameter;
	fbRegister: FB_IPCDiag_Register;
END_VAR
VAR // added by the converter: edge detectors and wires of the graphical bodies
    _w1, _w2 : BOOL;
END_VAR

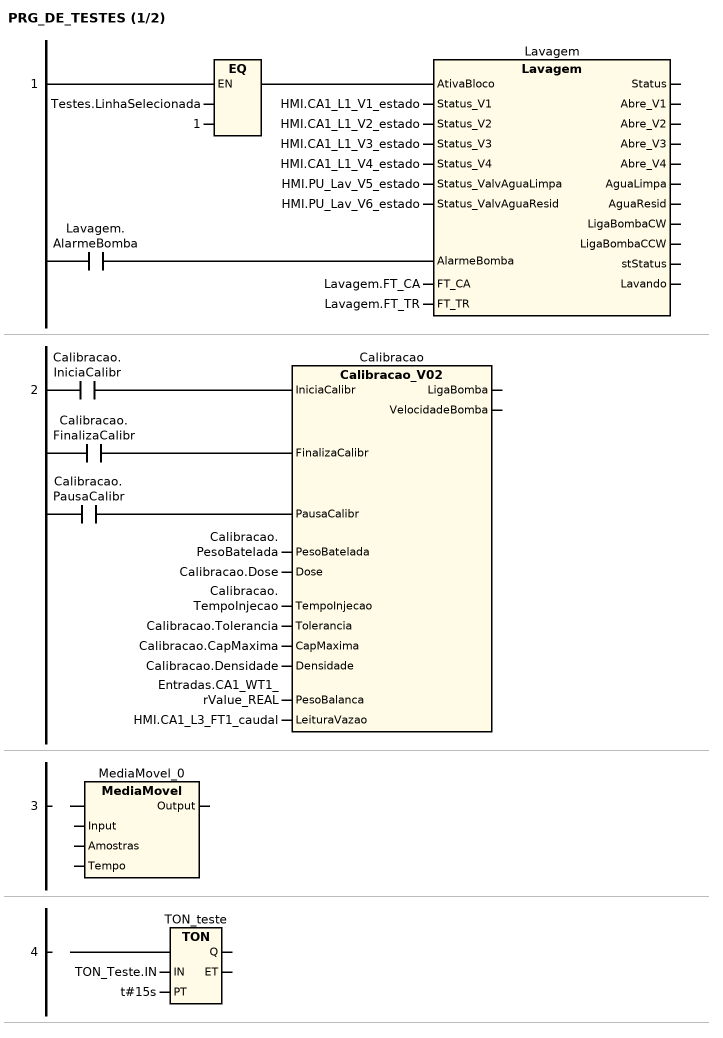
// NETWORK 1
Lavagem(
    AtivaBloco := Testes.LinhaSelecionada = 1,
    Status_V1 := HMI.CA1_L1_V1_estado,
    Status_V2 := HMI.CA1_L1_V2_estado,
    Status_V3 := HMI.CA1_L1_V3_estado,
    Status_V4 := HMI.CA1_L1_V4_estado,
    Status_ValvAguaLimpa := HMI.PU_Lav_V5_estado,
    Status_ValvAguaResid := HMI.PU_Lav_V6_estado,
    AlarmeBomba := Lavagem.AlarmeBomba,
    FT_CA := Lavagem.FT_CA,
    FT_TR := Lavagem.FT_TR);

// NETWORK 2
Calibracao(
    IniciaCalibr := Calibracao.IniciaCalibr,
    FinalizaCalibr := Calibracao.FinalizaCalibr,
    PausaCalibr := Calibracao.PausaCalibr,
    PesoBatelada := Calibracao.PesoBatelada,
    Dose := Calibracao.Dose,
    TempoInjecao := Calibracao.TempoInjecao,
    Tolerancia := Calibracao.Tolerancia,
    CapMaxima := Calibracao.CapMaxima,
    Densidade := Calibracao.Densidade,
    PesoBalanca := Entradas.CA1_WT1_rValue_REAL,
    LeituraVazao := HMI.CA1_L3_FT1_caudal); // Calibracao_V02

// NETWORK 3
MediaMovel_0(); // MediaMovel

// NETWORK 4
TON_teste(IN := TON_Teste.IN, PT := t#15s); // TON

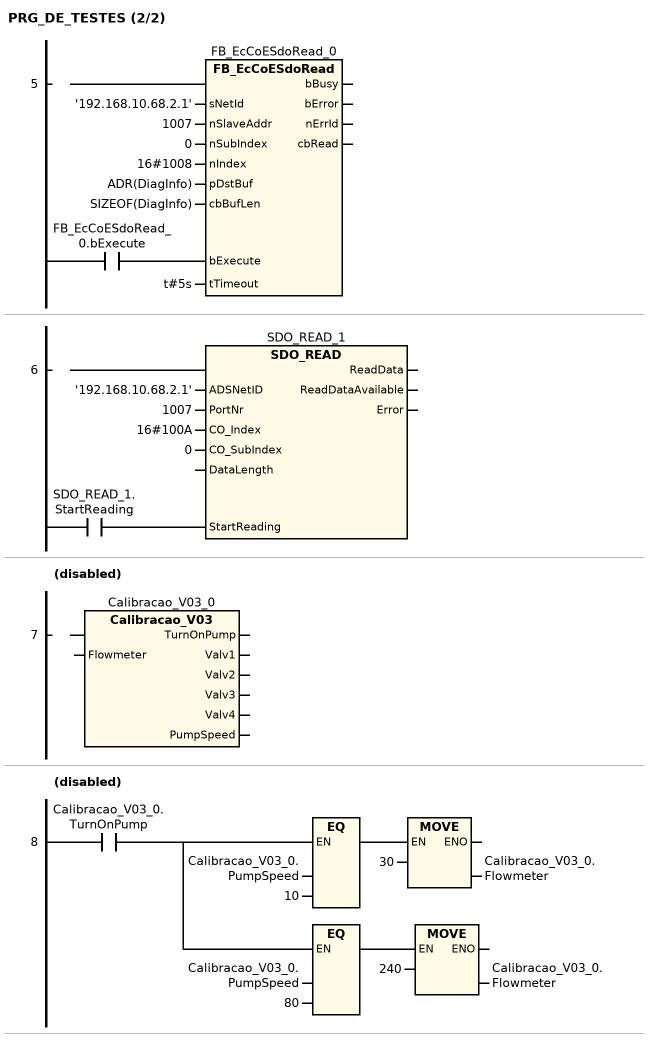
// NETWORK 5
FB_EcCoESdoRead_0(
    sNetId := '192.168.10.68.2.1',
    nSlaveAddr := 1007,
    nSubIndex := 0,
    nIndex := 16#1008,
    pDstBuf := ADR(DiagInfo),
    cbBufLen := SIZEOF(DiagInfo),
    bExecute := FB_EcCoESdoRead_0.bExecute,
    tTimeout := t#5s); // FB_EcCoESdoRead

// NETWORK 6
SDO_READ_1(
    ADSNetID := '192.168.10.68.2.1',
    PortNr := 1007,
    CO_Index := 16#100A,
    CO_SubIndex := 0,
    StartReading := SDO_READ_1.StartReading); // SDO_READ

// NETWORK 7 (disabled)
// Calibracao_V03_0(); // Calibracao_V03

// NETWORK 8 (disabled)
// _w1 := Calibracao_V03_0.TurnOnPump AND Calibracao_V03_0.PumpSpeed = 10;
// IF _w1 THEN Calibracao_V03_0.Flowmeter := 30; END_IF
// _w2 := Calibracao_V03_0.TurnOnPump AND Calibracao_V03_0.PumpSpeed = 80;
// IF _w2 THEN Calibracao_V03_0.Flowmeter := 240; END_IF

END_PROGRAM

// ---- POUs/Testes Thiago/Calibracao_V02.TcPOU
FUNCTION_BLOCK Calibracao_V02
VAR_INPUT
	//Comandos
	IniciaCalibr	:BOOL;	//Inicia processo de calibração
	FinalizaCalibr	:BOOL;	//Finaliza calibração
	PausaCalibr		:BOOL;	//Pausa calibração
	
	//Parâmetros inseridos pelo usuário
	PesoBatelada	:REAL;	//Peso da batelada					(kg)
	Dose		:REAL;	//Dose de produto a cada 100 kg		(mL/100 kg)
	TempoInjecao	:DINT;	//Tempo de injeção de produto		(s)
	Tolerancia		:REAL;	//Tolerância a erros				(%)
	CapMaxima		:REAL;	//Capacidade máxima do recipiente	(L)
	Densidade		:REAL;	//Densidade do produto				(kg/L)
	
	//Leituras externas
	PesoBalanca		:REAL;	//Peso da balança					(kg)
	LeituraVazao	:REAL;	//Valor vindo do sensor de vazão	(L/min)
END_VAR
VAR_OUTPUT
	LigaBomba		:BOOL;	//Saída para ligar a bomba
	VelocidadeBomba	:LREAL;	//Velocidade enviada para a bomba	(%)
END_VAR
VAR
	PID_BombaInjecao	:FB_BasicPID;	//PID Para controle da bomba de injeção
	Status				:INT;
	SwitchCase			:INT := 0;
	VolRecipiente		:REAL;	//Volume que deve ter no recipiente após a injeção
	TaraBalanca			:REAL;
	VazaoTotalizada		:REAL;	//Vazão do sensor totalizada
	Totalizar			:BOOL;	//Se verdadeiro, o totalizador deve ser ativado
	PulsosDoTotalizador	:REAL;	//Pulsos que o totalizador deu. Necessário para calcular a vazão média
	UltimasCalibr		:ARRAY [1..10] OF REAL;	//Array com as últimas calibrações
	IndexCalibr			:INT := 0;	//Index para o array de calibrações
	VelocEncontrada		:LREAL;	//Velocidade encontrada pela calibração
	
	iCounter			:INT;	// Variável de iteração do FOR
	SP_VazaoMedia		:REAL;	// Setpoint de vazão média para atingir o objetivo de dosagem
	PV_VazaoMedia		:REAL;	// Vazão média, calculada pela vazão e tempo de aplicação atual
	TON_TempoInjecao	:TON;	//Tempo de injeção
	TON_Totalizador		:TON;	//Temporizador para o totalizador de vazão
	CalibrSucesso		:BOOL;	// Calibração feita com sucesso
	
	Tara				:REAL; //Valor da tara da baalança
	TON_EntreCalibracoes: TON;
END_VAR

//Status da calibração
IF PesoBatelada <= 0 THEN
	Status := 1;	//Ajustar peso da batelada
ELSIF Dose <= 0 THEN
	Status := 2;	//Ajustar dosagem
ELSIF TempoInjecao <= 0 THEN
	Status := 3;	//Ajustar tempo de injeção
ELSIF Tolerancia <= 0 THEN
	Status := 4;	//Ajustar tolerância de erro
ELSIF CapMaxima <= 0 THEN
	Status := 5;	//Ajustar capacidade máxima
ELSIF Densidade <= 0 THEN
	Status := 6;	//Ajustar densidade do produto
ELSIF PausaCalibr THEN
	Status := 7;	//Calibração pausada
ELSIF SwitchCase > 0 THEN
	Status := 8;	//Calibrando
ELSIF (PesoBalanca/Densidade) > 0.9 * CapMaxima THEN
	Status := 9;	//Balança cheia
ELSIF ((PesoBatelada*Dose)/100)/1000 + (PesoBalanca/Densidade) > 0.9 * CapMaxima THEN
	Status := 10;	//Próxima aplicação irá transbordar o recipiente
ELSE
	Status := 99;	//Pronto para calibrar
END_IF

//Quando for fazer o teste, tentar aumentar o tempo de dosagem, já que a bomba vai buscar a vazão média, não importa o tempo de dosagem

//Instância dos temporizadores
TON_TempoInjecao(IN:= , PT:= DINT_TO_TIME(TempoInjecao*1000), Q=> , ET=> ); //Mult. por 1000 pois o timer recebe o valor em ms
TON_Totalizador(IN:= Totalizar AND NOT TON_Totalizador.Q, PT:= T#1S, Q=> , ET=> );
TON_EntreCalibracoes(IN:= , PT:= T#5S, Q=> , ET=> );

//Inicia a calibração
IF Status = 99 AND IniciaCalibr THEN
	Tara := PesoBalanca;
	SwitchCase := 5;
	IniciaCalibr := FALSE;
END_IF

//Finaliza a calibração
IF FinalizaCalibr THEN
	SwitchCase := 0;
	FinalizaCalibr := FALSE;
END_IF

//Totalizador de vazão
IF TON_Totalizador.Q THEN
	VazaoTotalizada := VazaoTotalizada + (LeituraVazao/60); //Dividido por 60 para converter de L/min para L/s;
	PulsosDoTotalizador := PulsosDoTotalizador + 1;
	PV_VazaoMedia := VazaoTotalizada/PulsosDoTotalizador;
END_IF

//Cálculo das variáveis usadas na calibração
VolRecipiente := (PesoBatelada*Dose)/100;	//É dividido por 100 por que a dosagem é a quantidade de mL a cada 100 kg
IF TempoInjecao <> 0 THEN
	SP_VazaoMedia := VolRecipiente/(DINT_TO_REAL(TempoInjecao)*1000); //É dividido por 100 para transformar de mL/s para L/s
END_IF

CASE SwitchCase OF
	0:	LigaBomba := FALSE;
		VelocidadeBomba := 0.0;
		PulsosDoTotalizador := 0;
		VazaoTotalizada := 0.0;
		Totalizar := FALSE;
		TON_TempoInjecao.IN := FALSE;
		IndexCalibr := 0;
		
	5:	FOR iCounter := 1 TO 10 BY 1 DO	//Limpa o array das ultimas calibrações
			UltimasCalibr[iCounter] := 0.0;
		END_FOR
		SwitchCase := 10;
		
	10:	IndexCalibr := IndexCalibr + 1;	//Incrementa o index do array de calibrações
		Totalizar := TRUE;
		SwitchCase := 20;
		
	20:	LigaBomba := TRUE;
		PID_BombaInjecao(
			fSetpointValue:= SP_VazaoMedia, 
			fActualValue:= PV_VazaoMedia, 
			bReset:= , 
			fCtrlCycleTime:= 0.1, 
			fKp:= 1, 
			fTn:= , 
			fTv:= , 
			fTd:= , 
			fCtrlOutput=> VelocidadeBomba, 
			nErrorStatus=> );
	PID_BombaInjecao.fTn := SEL(PID_BombaInjecao.fCtrlOutput > 150, 0.1, 0);

			
		TON_TempoInjecao.IN := TRUE;
		IF TON_TempoInjecao.Q THEN
			SwitchCase := 30;
			VelocEncontrada := VelocidadeBomba;
			LigaBomba := FALSE;
			TON_TempoInjecao.IN := FALSE;
		END_IF
		
	30:	//Aguarda confirmação de calibração bem sucedida
		UltimasCalibr[IndexCalibr] := (PesoBalanca - Tara)/Densidade;	//Fazer tara da balança se for necessário outra calibração
		
		//Calibração fora da tolerância
		IF UltimasCalibr[IndexCalibr] < VolRecipiente * (100 - Tolerancia)/100 OR UltimasCalibr[IndexCalibr] > VolRecipiente * (100 + Tolerancia)/100 THEN
			TON_EntreCalibracoes.IN := TRUE;
			IF TON_EntreCalibracoes.Q THEN
				TON_EntreCalibracoes.IN := FALSE;
				Tara := PesoBalanca;
				SwitchCase := 10;
			END_IF
			
		ELSE
				CalibrSucesso := TRUE;
				SwitchCase := 0;
		END_IF
		
		
END_CASE



(*----SIMULAÇÃO----*)

END_FUNCTION_BLOCK

// ---- POUs/Testes Thiago/MediaMovel.TcPOU
FUNCTION_BLOCK MediaMovel
VAR_INPUT
	Input		:REAL;	//Valor de entrada para fazer a média
	Amostras	:INT;	//Quantidade de amostras do valor de entrada para fazer a média móvel
	Tempo		:DINT;	//Tempo de amostragem
END_VAR
VAR_OUTPUT
	Output	:REAL;	//Valor da média móvel
END_VAR
VAR
	ArrayValores	:ARRAY[0..100] OF REAL;
	iCounter: INT;
	Acumulador: REAL;
	TON_TempoAmostra: TON;
END_VAR

//Se a quantidade de amostras for menor que 1, esse valor é configurado
IF Amostras < 1 THEN
	Amostras := 1;
ELSIF Amostras > 100 THEN
	Amostras := 100;
END_IF

//Temporizador para amostragem
TON_TempoAmostra(IN:= NOT TON_TempoAmostra.Q, PT:= DINT_TO_TIME(Tempo * 1000), Q=> , ET=> );

IF TON_TempoAmostra.Q THEN
	FOR iCounter := 1 TO (Amostras - 1) BY 1 DO
		ArrayValores[iCounter] := ArrayValores[iCounter + 1];
	END_FOR
	ArrayValores[Amostras] := Input;
END_IF

//Acumula os valores do array
Acumulador := 0;
FOR iCounter := 1 TO Amostras BY 1 DO
	Acumulador := Acumulador + ArrayValores[iCounter];
END_FOR

//Calcula a saída
Output := Acumulador / Amostras;

END_FUNCTION_BLOCK

// ---- POUs/Testes Thiago/CalculoConsumo.TcPOU
PROGRAM CalculoConsumo
VAR
	TON_CalculoConsumo	:TON;
	ResetConsumo		:BOOL;	//Reseta os dados de consumo
	DiaAtual			:WORD;
	iCounter: INT;
	iCounter2: INT;
	Teste: BOOL;
	i: INT;
	// Borda de início de tratamento
	InicioTrat: R_TRIG;
	Teste2: TIME;
END_VAR
VAR PERSISTENT
	Consumos		:ARRAY[1..12] OF REAL;	//Array com os consumos atuais
	UltimosDias		:ARRAY[1..12] OF ARRAY[1..30] OF REAL;
	RTRIG_Reset		:R_TRIG;
END_VAR

//Essa rotina calcula o consumo do uso de cada linha de acordo com o primeiro sensor de vazão


TON_CalculoConsumo(IN:=TRUE AND NOT TON_CalculoConsumo.Q, PT:=T#1S); //Pulsa a cada 1s

IF TON_CalculoConsumo.Q THEN
	//Os dados são divididos por 1000 para converter a vazão de mL/s para L/s. Só a vazão positiva é contabilizada
	//Totem 1
	DatosProceso.ConsumoCircuito_1 := DatosProceso.ConsumoCircuito_1 + SEL(HMI.CA1_L1_FT1_caudal/1000 > 0, 0, HMI.CA1_L1_FT1_caudal/1000);
	DatosProceso.ConsumoCircuito_2 := DatosProceso.ConsumoCircuito_2 + SEL(HMI.CA1_L2_FT1_caudal/1000 > 0, 0, HMI.CA1_L2_FT1_caudal/1000);
	DatosProceso.ConsumoCircuito_3 := DatosProceso.ConsumoCircuito_3 + SEL(HMI.CA1_L3_FT1_caudal/1000 > 0, 0, HMI.CA1_L3_FT1_caudal/1000);
	DatosProceso.ConsumoCircuito_4 := DatosProceso.ConsumoCircuito_4 + SEL(HMI.CA1_L4_FT1_caudal/1000 > 0, 0, HMI.CA1_L4_FT1_caudal/1000);
	Consumos[1] := Consumos[1] + SEL(HMI.CA1_L1_FT1_caudal > 0, 0, HMI.CA1_L1_FT1_caudal/1000);
	Consumos[2] := Consumos[2] + SEL(HMI.CA1_L2_FT1_caudal > 0, 0, HMI.CA1_L1_FT1_caudal/1000);
	Consumos[3] := Consumos[3] + SEL(HMI.CA1_L3_FT1_caudal > 0, 0, HMI.CA1_L1_FT1_caudal/1000);
	Consumos[4] := Consumos[4] + SEL(HMI.CA1_L4_FT1_caudal > 0, 0, HMI.CA1_L1_FT1_caudal/1000);
	
	//Totem 2
	DatosProceso.ConsumoCircuito_5 := DatosProceso.ConsumoCircuito_5 + SEL(HMI.CA2_L5_FT1_caudal/1000 > 0, 0, HMI.CA2_L5_FT1_caudal/1000);
	DatosProceso.ConsumoCircuito_6 := DatosProceso.ConsumoCircuito_6 + SEL(HMI.CA2_L6_FT1_caudal/1000 > 0, 0, HMI.CA2_L6_FT1_caudal/1000);
	DatosProceso.ConsumoCircuito_7 := DatosProceso.ConsumoCircuito_7 + SEL(HMI.CA2_L7_FT1_caudal/1000 > 0, 0, HMI.CA2_L7_FT1_caudal/1000);
	DatosProceso.ConsumoCircuito_8 := DatosProceso.ConsumoCircuito_8 + SEL(HMI.CA2_L8_FT1_caudal/1000 > 0, 0, HMI.CA2_L8_FT1_caudal/1000);
	Consumos[5] := Consumos[5] + SEL(HMI.CA2_L5_FT1_caudal > 0, 0, HMI.CA2_L5_FT1_caudal/1000);
	Consumos[6] := Consumos[6] + SEL(HMI.CA2_L6_FT1_caudal > 0, 0, HMI.CA2_L6_FT1_caudal/1000);
	Consumos[7] := Consumos[7] + SEL(HMI.CA2_L7_FT1_caudal > 0, 0, HMI.CA2_L7_FT1_caudal/1000);
	Consumos[8] := Consumos[8] + SEL(HMI.CA2_L8_FT1_caudal > 0, 0, HMI.CA2_L8_FT1_caudal/1000);
	
	//Totem 3
	DatosProceso.ConsumoCircuito_9 := DatosProceso.ConsumoCircuito_9 + SEL(HMI.CA3_L9_FT1_caudal/1000 > 0, 0, HMI.CA3_L9_FT1_caudal/1000);
	DatosProceso.ConsumoCircuito_10 := DatosProceso.ConsumoCircuito_10 + SEL(HMI.CA3_L10_FT1_caudal/1000 > 0, 0, HMI.CA3_L10_FT1_caudal/1000);
	DatosProceso.ConsumoCircuito_11 := DatosProceso.ConsumoCircuito_11 + SEL(HMI.CA3_L11_FT1_caudal/1000 > 0, 0, HMI.CA3_L11_FT1_caudal/1000);
	DatosProceso.ConsumoCircuito_12 := DatosProceso.ConsumoCircuito_12 + SEL(HMI.CA3_L12_FT1_caudal/1000 > 0, 0, HMI.CA3_L12_FT1_caudal/1000);
	Consumos[9] := Consumos[9] + SEL(HMI.CA3_L9_FT1_caudal > 0, 0, HMI.CA3_L9_FT1_caudal/1000);
	Consumos[10] := Consumos[10] + SEL(HMI.CA3_L10_FT1_caudal > 0, 0, HMI.CA3_L10_FT1_caudal/1000);
	Consumos[11] := Consumos[11] + SEL(HMI.CA3_L11_FT1_caudal > 0, 0, HMI.CA3_L11_FT1_caudal/1000);
	Consumos[12] := Consumos[12] + SEL(HMI.CA3_L12_FT1_caudal > 0, 0, HMI.CA3_L12_FT1_caudal/1000);
	
END_IF

RTRIG_Reset(CLK:=DatosProceso.LoteCargado);

IF ResetConsumo OR RTRIG_Reset.Q THEN
	DatosProceso.ConsumoCircuito_1 := 0;
	DatosProceso.ConsumoCircuito_2 := 0;
	DatosProceso.ConsumoCircuito_3 := 0;
	DatosProceso.ConsumoCircuito_4 := 0;
	DatosProceso.ConsumoCircuito_5 := 0;
	DatosProceso.ConsumoCircuito_6 := 0;
	DatosProceso.ConsumoCircuito_7 := 0;
	DatosProceso.ConsumoCircuito_8 := 0;
	DatosProceso.ConsumoCircuito_9 := 0;
	DatosProceso.ConsumoCircuito_10 := 0;
	DatosProceso.ConsumoCircuito_11 := 0;
	DatosProceso.ConsumoCircuito_12 := 0;
	DatosProceso.ConsumoPolvo_1 := 0;
	DatosProceso.ConsumoPolvo_2 := 0;
	FOR i := 1 TO 12 DO
		Consumos[i] := 0;
	END_FOR
	ResetConsumo := FALSE;
END_IF

IF DiaAtual <> Main.fbTime.systemTime.wDay THEN
	FOR iCounter := 1 TO 12 BY 1 DO
		//Faz o shift do array
		FOR iCounter2 := 1 TO 29 BY 1 DO
			UltimosDias[iCounter][iCounter2] := UltimosDias[iCounter][iCounter2 + 1];
		END_FOR
		UltimosDias[iCounter][30] := Consumos[iCounter];	//Transfere o consumo para o array de histórico
		Consumos[iCounter] := 0;							//Zera o array de consumo
	END_FOR
	DiaAtual := Main.fbTime.systemTime.wDay;
	//Teste := FALSE;
END_IF

//Computa a data e hora do inicio do tratamento atual
InicioTrat(CLK := HMI.bRun OR Teste);

IF InicioTrat.Q THEN
	DatosProceso.InicioTratamento := DT_TO_UDINT(MAIN.HoraAtual);
END_IF


//Cálculo do tempo restante para tratar todo o lote. 
DatosProceso.TempoRestante := SEL(DatosProceso.KgLote_Procesados > 0 AND (HMI.bRun OR Teste) AND DatosProceso.Kg_a_Procesar > DatosProceso.KgLote_Procesados, 0,(DatosProceso.Kg_a_Procesar/DatosProceso.KgLote_Procesados) * (DT_TO_UDINT(MAIN.HoraAtual) - DatosProceso.InicioTratamento));

//Cálculo do tempo decorrido no tratamento atual
DatosProceso.TempoTratamento := SEL(HMI.bRun OR Teste, 0, (DT_TO_UDINT(MAIN.HoraAtual) - DatosProceso.InicioTratamento));

//Cálculo do tempo total da batelada
DatosProceso.TempoTotal := SEL(DatosProceso.KgLote_Procesados > 0 AND(HMI.bRun OR Teste), 0, DatosProceso.TempoRestante + TO_REAL(DatosProceso.TempoTratamento));

Teste2 := REAL_TO_TIME(DatosProceso.TempoRestante*1000);

END_PROGRAM

// ---- POUs/Testes Thiago/ConsumoIBCs.TcPOU
PROGRAM ConsumoIBCs
VAR PERSISTENT
	ConsumoDiario	:ARRAY[1..12] OF REAL;	//Array com o consumo diário do IBC
	ConsumoSemanal	:ARRAY[1..12] OF REAL;	//Array com o consumo semanal do IBC
	ConsumoMensal	:ARRAY[1..12] OF REAL;	//Array com o consumo mensal do IBC
	ValorAtual		:ARRAY[1..12] OF REAL;	//Valor atual do IBC
	ValorInicial	:ARRAY[1..12] OF REAL;	//Peso dos IBCs no inicio do dia
	UltimosDias		:ARRAY[1..12] OF ARRAY[1..30] OF REAL;	//Array com o consumo dos últimos 30 dias
	
	DiaAtual	:WORD;
	SemanaAtual	:WORD;
	MesAtual	:WORD;
	
	Reabastecimento	:ARRAY[1..12] OF REAL;	//Essa variável é usada para detectar se o IBC foi abastecido
	
	//Configurações da média móvel
	Amostras	:INT;	//Quantidade de amostras
	Tempo		:DINT;	//Tempo de amostragem (s)
END_VAR

VAR
	iCounter: INT;
	TON_ConsumoIBC: TON;
	VarAux	:ARRAY[1..12] OF REAL;
	MediaM	:ARRAY[1..12] OF MediaMovel;
	iCounter2: INT;
	Teste: BOOL;
END_VAR

//Esse programa calcula o consumo diário dos IBCs
MediaM[1](Input:= , Amostras:= , Tempo:= , Output=> );

Amostras	:= 10;
Tempo		:= 2;
//Salva os valores atuais dos IBCs no array já com a média móvel aplicada
MediaM[1](Input:=Entradas.PU1_WT1_rValue_REAL, Amostras:= Amostras, Tempo:= Tempo, Output=> ValorAtual[1]);
MediaM[2](Input:=Entradas.PU1_WT2_rValue_REAL, Amostras:= Amostras, Tempo:= Tempo, Output=> ValorAtual[2]);
MediaM[3](Input:=Entradas.PU1_WT3_rValue_REAL, Amostras:= Amostras, Tempo:= Tempo, Output=> ValorAtual[3]);
MediaM[4](Input:=Entradas.PU1_WT4_rValue_REAL, Amostras:= Amostras, Tempo:= Tempo, Output=> ValorAtual[4]);
MediaM[5](Input:=Entradas.PU2_WT5_rValue_REAL, Amostras:= Amostras, Tempo:= Tempo, Output=> ValorAtual[5]);
MediaM[6](Input:=Entradas.PU2_WT6_rValue_REAL, Amostras:= Amostras, Tempo:= Tempo, Output=> ValorAtual[6]);
MediaM[7](Input:=Entradas.PU2_WT7_rValue_REAL, Amostras:= Amostras, Tempo:= Tempo, Output=> ValorAtual[7]);
MediaM[8](Input:=Entradas.PU2_WT8_rValue_REAL, Amostras:= Amostras, Tempo:= Tempo, Output=> ValorAtual[8]);
MediaM[9](Input:=Entradas.PU3_WT9_rValue_REAL, Amostras:= Amostras, Tempo:= Tempo, Output=> ValorAtual[9]);
MediaM[10](Input:=Entradas.PU3_WT10_rValue_REAL, Amostras:= Amostras, Tempo:= Tempo, Output=> ValorAtual[10]);
MediaM[11](Input:=Entradas.PU3_WT11_rValue_REAL, Amostras:= Amostras, Tempo:= Tempo, Output=> ValorAtual[11]);
MediaM[12](Input:=Entradas.PU3_WT12_rValue_REAL, Amostras:= Amostras, Tempo:= Tempo, Output=> ValorAtual[12]);

//Ao trocar o dia, o cálculo é zerado
IF DiaAtual <> Main.fbTime.systemTime.wDay OR Teste THEN
	FOR iCounter := 1 TO 12 BY 1 DO
		//Faz o shift no array dos consumos dos ultimos dias
		FOR iCounter2 := 1 TO 29 BY 1 DO
			UltimosDias[iCounter][iCounter2] := UltimosDias[iCounter][iCounter2 + 1];
		END_FOR
		
		//Salva o consumo do dia na ultima posição do array de histórico
		UltimosDias[iCounter][30] := ConsumoDiario[iCounter];
		
		ConsumoDiario[iCounter] := 0;						//Zera o array de consumo diário
		VarAux[iCounter]		:= ValorAtual[iCounter];	//Configura o array auxiliar
	END_FOR
	
	//Configura o valor inicial dos IBCs
	ValorInicial[1] := Entradas.PU1_WT1_rValue_REAL;
	ValorInicial[2] := Entradas.PU1_WT2_rValue_REAL;
	ValorInicial[3] := Entradas.PU1_WT3_rValue_REAL;
	ValorInicial[4] := Entradas.PU1_WT4_rValue_REAL;
	ValorInicial[5] := Entradas.PU2_WT5_rValue_REAL;
	ValorInicial[6] := Entradas.PU2_WT6_rValue_REAL;
	ValorInicial[7] := Entradas.PU2_WT7_rValue_REAL;
	ValorInicial[8] := Entradas.PU2_WT8_rValue_REAL;
	ValorInicial[9] := Entradas.PU3_WT9_rValue_REAL;
	ValorInicial[10] := Entradas.PU3_WT9_rValue_REAL;
	ValorInicial[11] := Entradas.PU3_WT9_rValue_REAL;
	ValorInicial[12] := Entradas.PU3_WT9_rValue_REAL;
	
	//Atualiza o dia atual
	DiaAtual := Main.fbTime.systemTime.wDay;
	Teste := FALSE;
END_IF


/////////////A VarAux, salvará a ultima subtração. Se a subtração atual for menor que a anterior, ocorreu abastecimento

//O cálculo do consumo ocorrerá a cada 1 minuto
TON_ConsumoIBC(IN:= NOT TON_ConsumoIBC.Q, PT:= T#1M, Q=> , ET=> );

IF TON_ConsumoIBC.Q THEN
	FOR iCounter := 1 TO 12 BY 1 DO
		IF ValorAtual[iCounter] < VarAux[iCounter] THEN
			ConsumoDiario[iCounter] := ConsumoDiario[iCounter] + (VarAux[iCounter] - ValorAtual[iCounter]);
		END_IF
		VarAux[iCounter] := ValorAtual[iCounter];
	END_FOR;
END_IF;

//ConsumoDiario[iCounter] := ValorInicial[iCounter] - ValorAtual[iCounter];

END_PROGRAM

// ---- POUs/Testes Thiago/ConfigBombas.TcPOU
PROGRAM ConfigBombas
VAR
	//Modelo padrão
	Apex10:DUT_cfgBombas;	//Parâmetros da Apex 10
	Apex15:DUT_cfgBombas;	//Parâmetros da Apex 15
	Apex20:DUT_cfgBombas;	//Parâmetros da Apex 20
	Apex28:DUT_cfgBombas;	//Parâmetros da Apex 28
	
	HmiModeloBomba		:INT;	//Modelo da bomba em edição, vindo da IHM
	LinhaSelecionada	:INT;	//Linha em que a bomba esta sendo editada
	Editar				:BOOL;	//Comando para editar os parâmetros
END_VAR
VAR PERSISTENT
	BD_L01	:DUT_cfgBombas;	//Bomba de dosagem da linha 1
	BD_L02	:DUT_cfgBombas;	//Bomba de dosagem da linha 2
	BD_L03	:DUT_cfgBombas;	//Bomba de dosagem da linha 3
	BD_L04	:DUT_cfgBombas;	//Bomba de dosagem da linha 4
	BD_L05	:DUT_cfgBombas;	//Bomba de dosagem da linha 5
	BD_L06	:DUT_cfgBombas;	//Bomba de dosagem da linha 6
	BD_L07	:DUT_cfgBombas;	//Bomba de dosagem da linha 7
	BD_L08	:DUT_cfgBombas;	//Bomba de dosagem da linha 8
	BD_L09	:DUT_cfgBombas;	//Bomba de dosagem da linha 9
	BD_L10	:DUT_cfgBombas;	//Bomba de dosagem da linha 10
	BD_L11	:DUT_cfgBombas;	//Bomba de dosagem da linha 11
	BD_L12	:DUT_cfgBombas;	//Bomba de dosagem da linha 12
END_VAR

//Essa rotina gerencia as configurações das bombas de dosagem de liquidos

{Region "Configurações dos modelos"}
	//Apex 10
	Apex10.Apex 		:= 10;
	Apex10.VazaoNominal	:= 36.667;		//Ajustar a vazão
	Apex10.BandaMorta	:= 5;
	Apex10.Kp			:= 0.1;
	Apex10.Ti			:= 100;
	Apex10.OutMax		:= 100;
	Apex10.OutMin		:= 0;
	Apex10.PvMax		:= 500;
	Apex10.PvMin		:= 0;
	
	//Apex 15
	Apex15.Apex 		:= 15;
	Apex15.VazaoNominal	:= 80.556;		//Ajustar a vazão
	Apex15.BandaMorta	:= 5;
	Apex15.Kp			:= 0.1;
	Apex15.Ti			:= 100;
	Apex15.OutMax		:= 100;
	Apex15.OutMin		:= 0;
	Apex15.PvMax		:= 500;
	Apex15.PvMin		:= 0;
	
	//Apex 20
	Apex20.Apex 		:= 20;
	Apex20.VazaoNominal	:= 140.277;		//Ajustar a vazão
	Apex20.BandaMorta	:= 5;
	Apex20.Kp			:= 0.1;
	Apex20.Ti			:= 100;
	Apex20.OutMax		:= 100;
	Apex20.OutMin		:= 0;
	Apex20.PvMax		:= 500;
	Apex20.PvMin		:= 0;
	
	//Apex 28
	Apex28.Apex 		:= 28;
	Apex28.VazaoNominal	:= 347.222;		//Ajustar a vazão
	Apex28.BandaMorta	:= 5;
	Apex28.Kp			:= 0.1;
	Apex28.Ti			:= 100;
	Apex28.OutMax		:= 100;
	Apex28.OutMin		:= 0;
	Apex28.PvMax		:= 500;
	Apex28.PvMin		:= 0;
{endregion}

IF Editar THEN
	CASE LinhaSelecionada OF
		1:	CASE HmiModeloBomba OF
				10:	BD_L01 := Apex10;
				15: BD_L01 := Apex15;
				20: BD_L01 := Apex20;
				28: BD_L01 := Apex28;
			END_CASE
			
		2:	CASE HmiModeloBomba OF
			10:	BD_L02 := Apex10;
			15: BD_L02 := Apex15;
			20: BD_L02 := Apex20;
			28: BD_L02 := Apex28;
		END_CASE
		
		3:	CASE HmiModeloBomba OF
			10:	BD_L03 := Apex10;
			15: BD_L03 := Apex15;
			20: BD_L03 := Apex20;
			28: BD_L03 := Apex28;
		END_CASE
		
		4:	CASE HmiModeloBomba OF
			10:	BD_L04 := Apex10;
			15: BD_L04 := Apex15;
			20: BD_L04 := Apex20;
			28: BD_L04 := Apex28;
		END_CASE
		
		5:	CASE HmiModeloBomba OF
			10:	BD_L05 := Apex10;
			15: BD_L05 := Apex15;
			20: BD_L05 := Apex20;
			28: BD_L05 := Apex28;
		END_CASE
		
		6:	CASE HmiModeloBomba OF
			10:	BD_L06 := Apex10;
			15: BD_L06 := Apex15;
			20: BD_L06 := Apex20;
			28: BD_L06 := Apex28;
		END_CASE
		
		7:	CASE HmiModeloBomba OF
			10:	BD_L07 := Apex10;
			15: BD_L07 := Apex15;
			20: BD_L07 := Apex20;
			28: BD_L07 := Apex28;
		END_CASE
		
		8:	CASE HmiModeloBomba OF
			10:	BD_L08 := Apex10;
			15: BD_L08 := Apex15;
			20: BD_L08 := Apex20;
			28: BD_L08 := Apex28;
		END_CASE
		
		9:	CASE HmiModeloBomba OF
			10:	BD_L09 := Apex10;
			15: BD_L09 := Apex15;
			20: BD_L09 := Apex20;
			28: BD_L09 := Apex28;
		END_CASE
		
		10:	CASE HmiModeloBomba OF
			10:	BD_L10 := Apex10;
			15: BD_L10 := Apex15;
			20: BD_L10 := Apex20;
			28: BD_L10 := Apex28;
		END_CASE
		
		11:	CASE HmiModeloBomba OF
			10:	BD_L11 := Apex10;
			15: BD_L11 := Apex15;
			20: BD_L11 := Apex20;
			28: BD_L11 := Apex28;
		END_CASE
		
		12:	CASE HmiModeloBomba OF
			10:	BD_L12 := Apex10;
			15: BD_L12 := Apex15;
			20: BD_L12 := Apex20;
			28: BD_L12 := Apex28;
		END_CASE
	END_CASE
	Editar := FALSE;
END_IF

END_PROGRAM

// ---- POUs/PrecargaLiqInyeccion.TcPOU
FUNCTION_BLOCK PrecargaLiqInyeccion
VAR_INPUT
	CaudalimetroSup:REAL;
	Precarga:BOOL;
	VeloBombaSolicitada:REAL;
END_VAR
VAR_OUTPUT
	MarchaBomba:BOOL;
	VelocidadBomba:REAL;
END_VAR
VAR
END_VAR

IF CaudalimetroSup<0 THEN
	MarchaBomba:=TRUE;
	ELSE
	MarchaBomba:=FALSE;	
END_IF

END_FUNCTION_BLOCK

// ---- POUs/Testes Thiago/Filtro.TcPOU
FUNCTION Filtro : REAL
VAR_INPUT
	Input:REAL;	//Entrada do sensor
	Tempo:DINT := 500;	//Tempo de amostragem
END_VAR
VAR
	Amostras:ARRAY[1..50] OF REAL;
	TON_Amostras:TON;
	i		:INT;	//Variável de iteração do FOR
	Soma 	:REAL;	//Somatório dos valores do array
	Teste: INT;
END_VAR

TON_Amostras(IN := NOT TON_Amostras.Q, PT:=DINT_TO_TIME(Tempo));

IF TON_Amostras.Q THEN
	//Faz o shift do array
	FOR i := 1 TO 49 DO
		Amostras[i] := Amostras[i + 1];
	END_FOR
	
	//Insere a leitura do sensor na última posição
	Amostras[50] := Input;
	
	//Soma os valores do array
	Soma := 0;
	FOR i := 1 TO 50 DO
		Soma := Soma + Amostras[i];
	END_FOR
	
	Filtro := Soma / 50;
	
END_IF

END_FUNCTION

// ---- POUs/Testes Thiago/BancoDeDados.TcPOU
PROGRAM BancoDeDados
VAR_INPUT
	InsertMarcha: InsertBD_Comandos;
	InsertParada: InsertBD_Comandos;
	ComandoSalvar:ARRAY[1..200] OF BOOL;
	bExecuteInsert		: BOOL; 
END_VAR
VAR
	Parte1Comandos	:STRING[100];
	Parte2Comandos	:STRING;
	Parte3Comandos	:STRING;
	RecordInsert	:FB_DBRecordInsert_EX;
	sCmdInsert		:T_MaxString;
	bInsertBusy		:BOOL;
	bInsertError	:BOOL;
	bInsertErrID	:UDINT;
	nRecords		:UDINT;
	
	Teste: BOOL;
END_VAR



//Código de erro 1142 - Usuário sem permissão para fazer o insert
//Código de erro 1146 - Tabela não encontrada
//Código de erro 1064 - Erro de sintaxe

//Pedaços do comando SQL para ficar melhor a montagem no uso delas
Parte1Comandos := 'INSERT INTO `comandos` (`comando`, `data_hora`, `usuario`, `serial_maquina`) VALUES (';
Parte2Comandos := CONCAT(', CURRENT_TIMESTAMP,$'', Main.NomeUsuario);
Parte3Comandos := CONCAT('$', $'', CONCAT(Main.SerialDaMaquina, '$')'));

RecordInsert(
	sNetID:= '127.0.0.1.1.1', //String containing the AMS network ID of the target device, at which the ADS command is directed.
	hDBID:= 1, // Indicates the ID of the database to be used.
	pCmdAddr:= ADR(sCmdInsert), //Pointer to the executing INSERT command
	cbCmdSize:= SIZEOF(sCmdInsert), //Indicates the length of the INSERT command.
	bExecute:= bExecuteInsert, 
	tTimeout:= T#5S, 
	bBusy=> bInsertBusy, 
	bError=> bInsertError, 
	nErrID=> bInsertErrID);
	

//----------------------- Comandos de funcionamento da máquina -----------------------//
{region "Comandos da máquina"}
//Marcha
bExecuteInsert := FALSE;
IF ComandoSalvar[1] THEN
	InsertMarcha(Insert:= TRUE, NomeComando:= 'MARCHA', InsertOut=> bExecuteInsert, Comando=> sCmdInsert);
	ComandoSalvar[1] := FALSE;
END_IF

//Parar
IF ComandoSalvar[2] THEN
	InsertParada(Insert:= TRUE, NomeComando:= 'PARADA', InsertOut=> bExecuteInsert, Comando=> sCmdInsert);
	ComandoSalvar[2] := FALSE;
END_IF

//Manual
IF ComandoSalvar[3] THEN
	InsertParada(Insert:= TRUE, NomeComando:= 'MAQ. EM MANUAL', InsertOut=> bExecuteInsert, Comando=> sCmdInsert);
	ComandoSalvar[3] := FALSE;
END_IF

//Auto
IF ComandoSalvar[4] THEN
	InsertParada(Insert:= TRUE, NomeComando:= 'MAQ. EM AUTOM.', InsertOut=> bExecuteInsert, Comando=> sCmdInsert);
	ComandoSalvar[4] := FALSE;
END_IF

//Fechar Ordem
IF ComandoSalvar[5] THEN
	InsertParada(Insert:= TRUE, NomeComando:= 'FECHAR ORDEM', InsertOut=> bExecuteInsert, Comando=> sCmdInsert);
	ComandoSalvar[5] := FALSE;
END_IF

//Aceitar lote
IF ComandoSalvar[6] THEN
	InsertParada(Insert:= TRUE, NomeComando:= 'ACEITAR LOTE', InsertOut=> bExecuteInsert, Comando=> sCmdInsert);
	ComandoSalvar[6] := FALSE;
END_IF

//Uma batelada
IF ComandoSalvar[7] THEN
	InsertParada(Insert:= TRUE, NomeComando:= 'UMA BATELADA', InsertOut=> bExecuteInsert, Comando=> sCmdInsert);
	ComandoSalvar[7] := FALSE;
END_IF

//Contínuo
IF ComandoSalvar[8] THEN
	InsertParada(Insert:= TRUE, NomeComando:= 'CONTÍNUO', InsertOut=> bExecuteInsert, Comando=> sCmdInsert);
	ComandoSalvar[8] := FALSE;
END_IF

//Pausa
IF ComandoSalvar[9] THEN
	InsertParada(Insert:= TRUE, NomeComando:= 'PAUSA', InsertOut=> bExecuteInsert, Comando=> sCmdInsert);
	ComandoSalvar[9] := FALSE;
END_IF
{endregion}


//----------------------- Acionamento manual das válvulas -----------------------//
{region "Válvulas Circuito 1"}
//------------------- Válvulas Circuito 1 -------------------//

//Circuito 1 Valvula 1 manual
IF ComandoSalvar[10] THEN
	InsertParada(Insert:= TRUE, NomeComando:= 'VALV. 1 CIRC. 1 MANUAL', InsertOut=> bExecuteInsert, Comando=> sCmdInsert);
	ComandoSalvar[10] := FALSE;
END_IF

//Circuito 1 Valvula 2 manual
IF ComandoSalvar[11] THEN
	InsertParada(Insert:= TRUE, NomeComando:= 'VALV. 2 CIRC. 1 MANUAL', InsertOut=> bExecuteInsert, Comando=> sCmdInsert);
	ComandoSalvar[11] := FALSE;
END_IF

//Circuito 1 Valvula 3 manual
IF ComandoSalvar[12] THEN
	InsertParada(Insert:= TRUE, NomeComando:= 'VALV. 3 CIRC. 1 MANUAL', InsertOut=> bExecuteInsert, Comando=> sCmdInsert);
	ComandoSalvar[12] := FALSE;
END_IF

//Circuito 1 Valvula 4 manual
IF ComandoSalvar[13] THEN
	InsertParada(Insert:= TRUE, NomeComando:= 'VALV. 4 CIRC. 1 MANUAL', InsertOut=> bExecuteInsert, Comando=> sCmdInsert);
	ComandoSalvar[13] := FALSE;
END_IF	  
{endregion}

{region "Válvulas Circuito 2"}
//------------------- Válvulas Circuito 2 -------------------//

//Circuito 2 Valvula 1 manual
IF ComandoSalvar[14] THEN
	InsertParada(Insert:= TRUE, NomeComando:= 'VALV. 1 CIRC. 2 MANUAL', InsertOut=> bExecuteInsert, Comando=> sCmdInsert);
	ComandoSalvar[14] := FALSE;
END_IF

//Circuito 2 Valvula 2 manual
IF ComandoSalvar[15] THEN
	InsertParada(Insert:= TRUE, NomeComando:= 'VALV. 2 CIRC. 2 MANUAL', InsertOut=> bExecuteInsert, Comando=> sCmdInsert);
	ComandoSalvar[15] := FALSE;
END_IF

//Circuito 2 Valvula 3 manual
IF ComandoSalvar[16] THEN
	InsertParada(Insert:= TRUE, NomeComando:= 'VALV. 3 CIRC. 2 MANUAL', InsertOut=> bExecuteInsert, Comando=> sCmdInsert);
	ComandoSalvar[16] := FALSE;
END_IF

//Circuito 2 Valvula 4 manual
IF ComandoSalvar[17] THEN
	InsertParada(Insert:= TRUE, NomeComando:= 'VALV. 4 CIRC. 2 MANUAL', InsertOut=> bExecuteInsert, Comando=> sCmdInsert);
	ComandoSalvar[17] := FALSE;
END_IF
{endregion}

{region "Válvulas Circuito 3"}
//------------------- Válvulas Circuito 3 -------------------//

//Circuito 3 Valvula 1 manual
IF ComandoSalvar[18] THEN
	InsertParada(Insert:= TRUE, NomeComando:= 'VALV. 1 CIRC. 3 MANUAL', InsertOut=> bExecuteInsert, Comando=> sCmdInsert);
	ComandoSalvar[18] := FALSE;
END_IF

//Circuito 3 Valvula 2 manual
IF ComandoSalvar[19] THEN
	InsertParada(Insert:= TRUE, NomeComando:= 'VALV. 2 CIRC. 3 MANUAL', InsertOut=> bExecuteInsert, Comando=> sCmdInsert);
	ComandoSalvar[19] := FALSE;
END_IF

//Circuito 3 Valvula 3 manual
IF ComandoSalvar[20] THEN
	InsertParada(Insert:= TRUE, NomeComando:= 'VALV. 3 CIRC. 3 MANUAL', InsertOut=> bExecuteInsert, Comando=> sCmdInsert);
	ComandoSalvar[20] := FALSE;
END_IF

//Circuito 3 Valvula 4 manual
IF ComandoSalvar[21] THEN
	InsertParada(Insert:= TRUE, NomeComando:= 'VALV. 4 CIRC. 3 MANUAL', InsertOut=> bExecuteInsert, Comando=> sCmdInsert);
	ComandoSalvar[21] := FALSE;
END_IF
{endregion}

{region "Válvulas Circuito 4"}
//------------------- Válvulas Circuito 4 -------------------//

//Circuito 4 Valvula 1 manual
IF ComandoSalvar[22] THEN
	InsertParada(Insert:= TRUE, NomeComando:= 'VALV. 1 CIRC. 4 MANUAL', InsertOut=> bExecuteInsert, Comando=> sCmdInsert);
	ComandoSalvar[22] := FALSE;
END_IF

//Circuito 4 Valvula 2 manual
IF ComandoSalvar[23] THEN
	InsertParada(Insert:= TRUE, NomeComando:= 'VALV. 2 CIRC. 4 MANUAL', InsertOut=> bExecuteInsert, Comando=> sCmdInsert);
	ComandoSalvar[23] := FALSE;
END_IF

//Circuito 4 Valvula 3 manual
IF ComandoSalvar[24] THEN
	InsertParada(Insert:= TRUE, NomeComando:= 'VALV. 3 CIRC. 4 MANUAL', InsertOut=> bExecuteInsert, Comando=> sCmdInsert);
	ComandoSalvar[24] := FALSE;
END_IF

//Circuito 4 Valvula 4 manual
IF ComandoSalvar[25] THEN
	InsertParada(Insert:= TRUE, NomeComando:= 'VALV. 4 CIRC. 4 MANUAL', InsertOut=> bExecuteInsert, Comando=> sCmdInsert);
	ComandoSalvar[25] := FALSE;
END_IF
{endregion}

{region "Válvulas Circuito 5"}
//------------------- Válvulas Circuito 5 -------------------//

//Circuito 5 Valvula 1 manual
IF ComandoSalvar[26] THEN
	InsertParada(Insert:= TRUE, NomeComando:= 'VALV. 1 CIRC. 5 MANUAL', InsertOut=> bExecuteInsert, Comando=> sCmdInsert);
	ComandoSalvar[26] := FALSE;
END_IF

//Circuito 5 Valvula 2 manual
IF ComandoSalvar[27] THEN
	InsertParada(Insert:= TRUE, NomeComando:= 'VALV. 2 CIRC. 5 MANUAL', InsertOut=> bExecuteInsert, Comando=> sCmdInsert);
	ComandoSalvar[27] := FALSE;
END_IF

//Circuito 5 Valvula 3 manual
IF ComandoSalvar[28] THEN
	InsertParada(Insert:= TRUE, NomeComando:= 'VALV. 3 CIRC. 5 MANUAL', InsertOut=> bExecuteInsert, Comando=> sCmdInsert);
	ComandoSalvar[28] := FALSE;
END_IF

//Circuito 5 Valvula 4 manual
IF ComandoSalvar[29] THEN
	InsertParada(Insert:= TRUE, NomeComando:= 'VALV. 4 CIRC. 5 MANUAL', InsertOut=> bExecuteInsert, Comando=> sCmdInsert);
	ComandoSalvar[29] := FALSE;
END_IF
{endregion}

{region "Válvulas Circuito 6"}
//------------------- Válvulas Circuito 6 -------------------//

//Circuito 6 Valvula 1 manual
IF ComandoSalvar[30] THEN
	InsertParada(Insert:= TRUE, NomeComando:= 'VALV. 1 CIRC. 6 MANUAL', InsertOut=> bExecuteInsert, Comando=> sCmdInsert);
	ComandoSalvar[30] := FALSE;
END_IF

//Circuito 6 Valvula 2 manual
IF ComandoSalvar[31] THEN
	InsertParada(Insert:= TRUE, NomeComando:= 'VALV. 2 CIRC. 6 MANUAL', InsertOut=> bExecuteInsert, Comando=> sCmdInsert);
	ComandoSalvar[31] := FALSE;
END_IF

//Circuito 6 Valvula 3 manual
IF ComandoSalvar[32] THEN
	InsertParada(Insert:= TRUE, NomeComando:= 'VALV. 3 CIRC. 6 MANUAL', InsertOut=> bExecuteInsert, Comando=> sCmdInsert);
	ComandoSalvar[32] := FALSE;
END_IF

//Circuito 6 Valvula 4 manual
IF ComandoSalvar[33] THEN
	InsertParada(Insert:= TRUE, NomeComando:= 'VALV. 4 CIRC. 6 MANUAL', InsertOut=> bExecuteInsert, Comando=> sCmdInsert);
	ComandoSalvar[33] := FALSE;
END_IF
{endregion}

{region "Válvulas Circuito 7"}
//------------------- Válvulas Circuito 7 -------------------//

//Circuito 7 Valvula 1 manual
IF ComandoSalvar[34] THEN
	InsertParada(Insert:= TRUE, NomeComando:= 'VALV. 1 CIRC. 7 MANUAL', InsertOut=> bExecuteInsert, Comando=> sCmdInsert);
	ComandoSalvar[34] := FALSE;
END_IF

//Circuito 7 Valvula 2 manual
IF ComandoSalvar[35] THEN
	InsertParada(Insert:= TRUE, NomeComando:= 'VALV. 2 CIRC. 7 MANUAL', InsertOut=> bExecuteInsert, Comando=> sCmdInsert);
	ComandoSalvar[35] := FALSE;
END_IF

//Circuito 7 Valvula 3 manual
IF ComandoSalvar[36] THEN
	InsertParada(Insert:= TRUE, NomeComando:= 'VALV. 3 CIRC. 7 MANUAL', InsertOut=> bExecuteInsert, Comando=> sCmdInsert);
	ComandoSalvar[36] := FALSE;
END_IF
	 
//Circuito 7 Valvula 4 manual
IF ComandoSalvar[37] THEN
	InsertParada(Insert:= TRUE, NomeComando:= 'VALV. 4 CIRC. 7 MANUAL', InsertOut=> bExecuteInsert, Comando=> sCmdInsert);
	ComandoSalvar[37] := FALSE;
END_IF
{endregion}

{region "Válvulas Circuito 8"}
//------------------- Válvulas Circuito 8 -------------------//

//Circuito 8 Valvula 1 manual
IF ComandoSalvar[38] THEN
	InsertParada(Insert:= TRUE, NomeComando:= 'VALV. 1 CIRC. 8 MANUAL', InsertOut=> bExecuteInsert, Comando=> sCmdInsert);
	ComandoSalvar[38] := FALSE;
END_IF

//Circuito 8 Valvula 2 manual
IF ComandoSalvar[39] THEN
	InsertParada(Insert:= TRUE, NomeComando:= 'VALV. 2 CIRC. 8 MANUAL', InsertOut=> bExecuteInsert, Comando=> sCmdInsert);
	ComandoSalvar[39] := FALSE;
END_IF

//Circuito 8 Valvula 3 manual
IF ComandoSalvar[40] THEN
	InsertParada(Insert:= TRUE, NomeComando:= 'VALV. 3 CIRC. 8 MANUAL', InsertOut=> bExecuteInsert, Comando=> sCmdInsert);
	ComandoSalvar[40] := FALSE;
END_IF

//Circuito 8 Valvula 4 manual
IF ComandoSalvar[41] THEN
	InsertParada(Insert:= TRUE, NomeComando:= 'VALV. 4 CIRC. 8 MANUAL', InsertOut=> bExecuteInsert, Comando=> sCmdInsert);
	ComandoSalvar[41] := FALSE;
END_IF
{endregion}
	 

{region "Válvulas Circuito 9"}
//------------------- Válvulas Circuito 9 -------------------//

//Circuito 9 Valvula 1 manual
IF ComandoSalvar[42] THEN
	InsertParada(Insert:= TRUE, NomeComando:= 'VALV. 1 CIRC. 9 MANUAL', InsertOut=> bExecuteInsert, Comando=> sCmdInsert);
	ComandoSalvar[42] := FALSE;
END_IF

//Circuito 9 Valvula 2 manual
IF ComandoSalvar[43] THEN
	InsertParada(Insert:= TRUE, NomeComando:= 'VALV. 2 CIRC. 9 MANUAL', InsertOut=> bExecuteInsert, Comando=> sCmdInsert);
	ComandoSalvar[43] := FALSE;
END_IF

//Circuito 9 Valvula 3 manual
IF ComandoSalvar[44] THEN
	InsertParada(Insert:= TRUE, NomeComando:= 'VALV. 3 CIRC. 9 MANUAL', InsertOut=> bExecuteInsert, Comando=> sCmdInsert);
	ComandoSalvar[44] := FALSE;
END_IF

//Circuito 9 Valvula 4 manual
IF ComandoSalvar[45] THEN
	InsertParada(Insert:= TRUE, NomeComando:= 'VALV. 4 CIRC. 9 MANUAL', InsertOut=> bExecuteInsert, Comando=> sCmdInsert);
	ComandoSalvar[45] := FALSE;
END_IF
{endregion}
	 

{region "Válvulas Circuito 10"}
//------------------- Válvulas Circuito 10 -------------------//

//Circuito 10 Valvula 1 manual
IF ComandoSalvar[46] THEN
	InsertParada(Insert:= TRUE, NomeComando:= 'VALV. 1 CIRC. 10 MANUAL', InsertOut=> bExecuteInsert, Comando=> sCmdInsert);
	ComandoSalvar[46] := FALSE;
END_IF

//Circuito 10 Valvula 2 manual
IF ComandoSalvar[47] THEN
	InsertParada(Insert:= TRUE, NomeComando:= 'VALV. 2 CIRC. 10 MANUAL', InsertOut=> bExecuteInsert, Comando=> sCmdInsert);
	ComandoSalvar[47] := FALSE;
END_IF

//Circuito 10 Valvula 3 manual
IF ComandoSalvar[48] THEN
	InsertParada(Insert:= TRUE, NomeComando:= 'VALV. 3 CIRC. 10 MANUAL', InsertOut=> bExecuteInsert, Comando=> sCmdInsert);
	ComandoSalvar[48] := FALSE;
END_IF

//Circuito 10 Valvula 4 manual
IF ComandoSalvar[49] THEN
	InsertParada(Insert:= TRUE, NomeComando:= 'VALV. 4 CIRC. 10 MANUAL', InsertOut=> bExecuteInsert, Comando=> sCmdInsert);
	ComandoSalvar[49] := FALSE;
END_IF
{endregion}
	 

{region "Válvulas Circuito 11"}
//------------------- Válvulas Circuito 11 -------------------//

//Circuito 11 Valvula 1 manual
IF ComandoSalvar[50] THEN
	InsertParada(Insert:= TRUE, NomeComando:= 'VALV. 1 CIRC. 11 MANUAL', InsertOut=> bExecuteInsert, Comando=> sCmdInsert);
	ComandoSalvar[50] := FALSE;
END_IF

//Circuito 11 Valvula 2 manual
IF ComandoSalvar[51] THEN
	InsertParada(Insert:= TRUE, NomeComando:= 'VALV. 2 CIRC. 11 MANUAL', InsertOut=> bExecuteInsert, Comando=> sCmdInsert);
	ComandoSalvar[51] := FALSE;
END_IF

//Circuito 11 Valvula 3 manual
IF ComandoSalvar[52] THEN
	InsertParada(Insert:= TRUE, NomeComando:= 'VALV. 3 CIRC. 11 MANUAL', InsertOut=> bExecuteInsert, Comando=> sCmdInsert);
	ComandoSalvar[52] := FALSE;
END_IF

//Circuito 11 Valvula 4 manual
IF ComandoSalvar[53] THEN
	InsertParada(Insert:= TRUE, NomeComando:= 'VALV. 4 CIRC. 11 MANUAL', InsertOut=> bExecuteInsert, Comando=> sCmdInsert);
	ComandoSalvar[53] := FALSE;
END_IF
{endregion}
	 

{region "Válvulas Circuito 12"}
//------------------- Válvulas Circuito 12 -------------------//

//Circuito 12 Valvula 1 manual
IF ComandoSalvar[54] THEN
	InsertParada(Insert:= TRUE, NomeComando:= 'VALV. 1 CIRC. 12 MANUAL', InsertOut=> bExecuteInsert, Comando=> sCmdInsert);
	ComandoSalvar[54] := FALSE;
END_IF

//Circuito 12 Valvula 2 manual
IF ComandoSalvar[55] THEN
	InsertParada(Insert:= TRUE, NomeComando:= 'VALV. 2 CIRC. 12 MANUAL', InsertOut=> bExecuteInsert, Comando=> sCmdInsert);
	ComandoSalvar[55] := FALSE;
END_IF

//Circuito 12 Valvula 3 manual
IF ComandoSalvar[56] THEN
	InsertParada(Insert:= TRUE, NomeComando:= 'VALV. 3 CIRC. 12 MANUAL', InsertOut=> bExecuteInsert, Comando=> sCmdInsert);
	ComandoSalvar[56] := FALSE;
END_IF

//Circuito 12 Valvula 4 manual
IF ComandoSalvar[57] THEN
	InsertParada(Insert:= TRUE, NomeComando:= 'VALV. 4 CIRC. 12 MANUAL', InsertOut=> bExecuteInsert, Comando=> sCmdInsert);
	ComandoSalvar[57] := FALSE;
END_IF
{endregion}


//-----------------------			Acionamento manual das válvulas de água			-----------------------//
{region "Válvulas de água"}
//Válvula de água limpa
IF ComandoSalvar[58] THEN
	InsertParada(Insert:= TRUE, NomeComando:= 'VALV. AGUA LIMPA MANUAL', InsertOut=> bExecuteInsert, Comando=> sCmdInsert);
	ComandoSalvar[58] := FALSE;
END_IF

//Válvula de água residual
IF ComandoSalvar[59] THEN
	InsertParada(Insert:= TRUE, NomeComando:= 'VALV. 4 AGUA RESID. MANUAL', InsertOut=> bExecuteInsert, Comando=> sCmdInsert);
	ComandoSalvar[59] := FALSE;
END_IF
{endregion}
	 

//-----------------------			Acionamento manual das bombas de dosagem		-----------------------//
{region "Bombas de dosagem"}
//Bomba da linha 1
IF ComandoSalvar[60] THEN
	InsertParada(Insert:= TRUE, NomeComando:= 'BOMBA DOSAD. 1 MANUAL', InsertOut=> bExecuteInsert, Comando=> sCmdInsert);
	ComandoSalvar[60] := FALSE;
END_IF	
//Bomba da linha 2 
IF ComandoSalvar[61] THEN
	InsertParada(Insert:= TRUE, NomeComando:= 'BOMBA DOSAD. 2 MANUAL', InsertOut=> bExecuteInsert, Comando=> sCmdInsert);
	ComandoSalvar[61] := FALSE;
END_IF	 
//Bomba da linha 3
IF ComandoSalvar[62] THEN
	InsertParada(Insert:= TRUE, NomeComando:= 'BOMBA DOSAD. 3 MANUAL', InsertOut=> bExecuteInsert, Comando=> sCmdInsert);
	ComandoSalvar[62] := FALSE;
END_IF	 
//Bomba da linha 4
IF ComandoSalvar[63] THEN
	InsertParada(Insert:= TRUE, NomeComando:= 'BOMBA DOSAD. 4 MANUAL', InsertOut=> bExecuteInsert, Comando=> sCmdInsert);
	ComandoSalvar[63] := FALSE;
END_IF	 
//Bomba da linha 5
IF ComandoSalvar[64] THEN
	InsertParada(Insert:= TRUE, NomeComando:= 'BOMBA DOSAD. 5 MANUAL', InsertOut=> bExecuteInsert, Comando=> sCmdInsert);
	ComandoSalvar[64] := FALSE;
END_IF	 
//Bomba da linha 6
IF ComandoSalvar[65] THEN
	InsertParada(Insert:= TRUE, NomeComando:= 'BOMBA DOSAD. 6 MANUAL', InsertOut=> bExecuteInsert, Comando=> sCmdInsert);
	ComandoSalvar[65] := FALSE;
END_IF	 
//Bomba da linha 7
IF ComandoSalvar[66] THEN
	InsertParada(Insert:= TRUE, NomeComando:= 'BOMBA DOSAD. 7 MANUAL', InsertOut=> bExecuteInsert, Comando=> sCmdInsert);
	ComandoSalvar[66] := FALSE;
END_IF	 
//Bomba da linha 8
IF ComandoSalvar[67] THEN
	InsertParada(Insert:= TRUE, NomeComando:= 'BOMBA DOSAD. 8 MANUAL', InsertOut=> bExecuteInsert, Comando=> sCmdInsert);
	ComandoSalvar[67] := FALSE;
END_IF	 
//Bomba da linha 9
IF ComandoSalvar[68] THEN
	InsertParada(Insert:= TRUE, NomeComando:= 'BOMBA DOSAD. 9 MANUAL', InsertOut=> bExecuteInsert, Comando=> sCmdInsert);
	ComandoSalvar[68] := FALSE;
END_IF	 
//Bomba da linha 10
IF ComandoSalvar[69] THEN
	InsertParada(Insert:= TRUE, NomeComando:= 'BOMBA DOSAD. 10 MANUAL', InsertOut=> bExecuteInsert, Comando=> sCmdInsert);
	ComandoSalvar[69] := FALSE;
END_IF	 
//Bomba da linha 11
IF ComandoSalvar[70] THEN
	InsertParada(Insert:= TRUE, NomeComando:= 'BOMBA DOSAD. 11 MANUAL', InsertOut=> bExecuteInsert, Comando=> sCmdInsert);
	ComandoSalvar[70] := FALSE;
END_IF	 
//Bomba da linha 12
IF ComandoSalvar[71] THEN
	InsertParada(Insert:= TRUE, NomeComando:= 'BOMBA DOSAD. 12 MANUAL', InsertOut=> bExecuteInsert, Comando=> sCmdInsert);
	ComandoSalvar[71] := FALSE;
END_IF
{endregion}

//-----------------------			Acionamento manual dos agitadores				-----------------------//
{region "Agitadores"}
//Agitador da linha 1
IF ComandoSalvar[72] THEN
	InsertParada(Insert:= TRUE, NomeComando:= 'AGITADOR 1 MANUAL', InsertOut=> bExecuteInsert, Comando=> sCmdInsert);
	ComandoSalvar[72] := FALSE;
END_IF
//Agitador da linha 2
IF ComandoSalvar[73] THEN
	InsertParada(Insert:= TRUE, NomeComando:= 'AGITADOR 2 MANUAL', InsertOut=> bExecuteInsert, Comando=> sCmdInsert);
	ComandoSalvar[73] := FALSE;
END_IF
//Agitador da linha 3
IF ComandoSalvar[74] THEN
	InsertParada(Insert:= TRUE, NomeComando:= 'AGITADOR 3 MANUAL', InsertOut=> bExecuteInsert, Comando=> sCmdInsert);
	ComandoSalvar[74] := FALSE;
END_IF
//Agitador da linha 4
IF ComandoSalvar[75] THEN
	InsertParada(Insert:= TRUE, NomeComando:= 'AGITADOR 4 MANUAL', InsertOut=> bExecuteInsert, Comando=> sCmdInsert);
	ComandoSalvar[75] := FALSE;
END_IF
//Agitador da linha 5
IF ComandoSalvar[76] THEN
	InsertParada(Insert:= TRUE, NomeComando:= 'AGITADOR 5 MANUAL', InsertOut=> bExecuteInsert, Comando=> sCmdInsert);
	ComandoSalvar[76] := FALSE;
END_IF
//Agitador da linha 6
IF ComandoSalvar[77] THEN
	InsertParada(Insert:= TRUE, NomeComando:= 'AGITADOR 6 MANUAL', InsertOut=> bExecuteInsert, Comando=> sCmdInsert);
	ComandoSalvar[77] := FALSE;
END_IF
//Agitador da linha 7
IF ComandoSalvar[78] THEN
	InsertParada(Insert:= TRUE, NomeComando:= 'AGITADOR 7 MANUAL', InsertOut=> bExecuteInsert, Comando=> sCmdInsert);
	ComandoSalvar[78] := FALSE;
END_IF
//Agitador da linha 8
IF ComandoSalvar[79] THEN
	InsertParada(Insert:= TRUE, NomeComando:= 'AGITADOR 8 MANUAL', InsertOut=> bExecuteInsert, Comando=> sCmdInsert);
	ComandoSalvar[79] := FALSE;
END_IF
//Agitador da linha 9
IF ComandoSalvar[80] THEN
	InsertParada(Insert:= TRUE, NomeComando:= 'AGITADOR 9 MANUAL', InsertOut=> bExecuteInsert, Comando=> sCmdInsert);
	ComandoSalvar[80] := FALSE;
END_IF
//Agitador da linha 10
IF ComandoSalvar[81] THEN
	InsertParada(Insert:= TRUE, NomeComando:= 'AGITADOR 10 MANUAL', InsertOut=> bExecuteInsert, Comando=> sCmdInsert);
	ComandoSalvar[81] := FALSE;
END_IF
//Agitador da linha 11
IF ComandoSalvar[82] THEN
	InsertParada(Insert:= TRUE, NomeComando:= 'AGITADOR 11 MANUAL', InsertOut=> bExecuteInsert, Comando=> sCmdInsert);
	ComandoSalvar[82] := FALSE;
END_IF
//Agitador da linha 12
IF ComandoSalvar[83] THEN
	InsertParada(Insert:= TRUE, NomeComando:= 'AGITADOR 12 MANUAL', InsertOut=> bExecuteInsert, Comando=> sCmdInsert);
	ComandoSalvar[83] := FALSE;
END_IF
{endregion}

